LIN {X 0,Y 616.016,Z 683.652,A -85,B 0,C 180,E1 29122.379,E2 29122.379} C_VEL
LIN {X 0,Y 617.28,Z 685.528,A -85,B 0,C 180,E1 29121.476,E2 29121.476} C_VEL
LIN {X 0,Y 619.5,Z 690.288,A -85,B 0,C 180,E1 29120.03,E2 29120.03} C_VEL
LIN {X 0,Y 621.765,Z 695.272,A -85,B 0,C 180,E1 29118.873,E2 29118.873} C_VEL
LIN {X 0,Y 624.795,Z 702.465,A -85,B 0,C 180,E1 29117.519,E2 29117.519} C_VEL
LIN {X 0,Y 628.158,Z 711.521,A -85,B 0,C 180,E1 29116.158,E2 29116.158} C_VEL
LIN {X 0,Y 622.39,Z 748.268,A -85,B 0,C 180,E1 29113.628,E2 29113.628} C_VEL
LIN {X 0,Y 618.399,Z 786.592,A -85,B 0,C 180,E1 29111.107,E2 29111.107} C_VEL
LIN {X 0,Y 618.395,Z 807.892,A -85,B 0,C 180,E1 29109.637,E2 29109.637} C_VEL
LIN {X 0,Y 620.24,Z 824.543,A -85,B 0,C 180,E1 29108.419,E2 29108.419} C_VEL
LIN {X 0,Y 623.991,Z 840.098,A -85,B 0,C 180,E1 29107.212,E2 29107.212} C_VEL
LIN {X 0,Y 629.828,Z 854.618,A -85,B 0,C 180,E1 29106.015,E2 29106.015} C_VEL
LIN {X 0,Y 636.961,Z 866.767,A -85,B 0,C 180,E1 29104.955,E2 29104.955} C_VEL
LIN {X 0,Y 645.236,Z 877.236,A -85,B 0,C 180,E1 29103.997,E2 29103.997} C_VEL
LIN {X 0,Y 655.85,Z 887.383,A -85,B 0,C 180,E1 29103.016,E2 29103.016} C_VEL
LIN {X 0,Y 667.322,Z 895.733,A -85,B 0,C 180,E1 29102.159,E2 29102.159} C_VEL
LIN {X 0,Y 672.025,Z 898.736,A -85,B 0,C 180,E1 29101.844,E2 29101.844} C_VEL
LIN {X 0,Y 649.338,Z 931.659,A -85,B 0,C 180,E1 29100.95,E2 29100.95} C_VEL
LIN {X 0,Y 638.123,Z 950.658,A -85,B 0,C 180,E1 29100.351,E2 29100.351} C_VEL
LIN {X 0,Y 630.355,Z 966.843,A -85,B 0,C 180,E1 29099.766,E2 29099.766} C_VEL
LIN {X 0,Y 626.313,Z 976.356,A -85,B 0,C 180,E1 29099.399,E2 29099.399} C_VEL
LIN {X 0,Y 619.977,Z 991.013,A -85,B 0,C 180,E1 29098.829,E2 29098.829} C_VEL
LIN {X 0,Y 614.207,Z 1008.828,A -85,B 0,C 180,E1 29098.082,E2 29098.082} C_VEL
LIN {X 0,Y 612.745,Z 1027.64,A -85,B 0,C 180,E1 29097.893,E2 29097.893} C_VEL
LIN {X 0,Y 612.102,Z 1064.345,A -85,B 0,C 180,E1 29097.385,E2 29097.385} C_VEL
LIN {X 0,Y 611.36,Z 1085.866,A -85,B 0,C 180,E1 29096.927,E2 29096.927} C_VEL
LIN {X 0,Y 610.423,Z 1107.35,A -85,B 0,C 180,E1 29096.299,E2 29096.299} C_VEL
LIN {X 0,Y 609.333,Z 1128.576,A -85,B 0,C 180,E1 29095.507,E2 29095.507} C_VEL
LIN {X 0,Y 608.179,Z 1148.795,A -85,B 0,C 180,E1 29094.577,E2 29094.577} C_VEL
LIN {X 0,Y 606.971,Z 1168.175,A -85,B 0,C 180,E1 29093.492,E2 29093.492} C_VEL
LIN {X 0,Y 605.739,Z 1186.859,A -85,B 0,C 180,E1 29092.26,E2 29092.26} C_VEL
LIN {X 0,Y 604.616,Z 1204.162,A -85,B 0,C 180,E1 29090.927,E2 29090.927} C_VEL
LIN {X 0,Y 603.528,Z 1220.54,A -85,B 0,C 180,E1 29089.45,E2 29089.45} C_VEL
LIN {X 0,Y 602.577,Z 1235.528,A -85,B 0,C 180,E1 29087.876,E2 29087.876} C_VEL
LIN {X 0,Y 601.792,Z 1249.417,A -85,B 0,C 180,E1 29086.186,E2 29086.186} C_VEL
LIN {X 0,Y 601.099,Z 1262.801,A -85,B 0,C 180,E1 29084.251,E2 29084.251} C_VEL
LIN {X 0,Y 600.679,Z 1273.278,A -85,B 0,C 180,E1 29082.496,E2 29082.496} C_VEL
LIN {X 0,Y 600.389,Z 1281.271,A -85,B 0,C 180,E1 29080.943,E2 29080.943} C_VEL
LIN {X 0,Y 600.168,Z 1289.619,A -85,B 0,C 180,E1 29079.008,E2 29079.008} C_VEL
LIN {X 0,Y 600.052,Z 1295.993,A -85,B 0,C 180,E1 29077.082,E2 29077.082} C_VEL
LIN {X 0,Y 599.998,Z 1300.183,A -85,B 0,C 180,E1 29075.449,E2 29075.449} C_VEL
LIN {X 0,Y 599.968,Z 1303.25,A -85,B 0,C 180,E1 29073.821,E2 29073.821} C_VEL
LIN {X 0,Y 599.962,Z 1305.145,A -85,B 0,C 180,E1 29072.291,E2 29072.291} C_VEL
LIN {X 0,Y 599.962,Z 1306.122,A -85,B 0,C 180,E1 29070.667,E2 29070.667} C_VEL
LIN {X 0,Y 599.969,Z 1306.047,A -85,B 0,C 180,E1 29069.044,E2 29069.044} C_VEL
LIN {X 0,Y 599.968,Z 1304.572,A -85,B 0,C 180,E1 29067.037,E2 29067.037} C_VEL
LIN {X 0,Y 599.975,Z 1301.11,A -85,B 0,C 180,E1 29064.931,E2 29064.931} C_VEL
LIN {X 0,Y 600.018,Z 1296.951,A -85,B 0,C 180,E1 29063.204,E2 29063.204} C_VEL
LIN {X 0,Y 600.122,Z 1291.846,A -85,B 0,C 180,E1 29061.568,E2 29061.568} C_VEL
LIN {X 0,Y 600.293,Z 1284.34,A -85,B 0,C 180,E1 29059.635,E2 29059.635} C_VEL
LIN {X 0,Y 600.621,Z 1274.844,A -85,B 0,C 180,E1 29057.695,E2 29057.695} C_VEL
LIN {X 0,Y 600.987,Z 1265.818,A -85,B 0,C 180,E1 29056.137,E2 29056.137} C_VEL
LIN {X 0,Y 601.5,Z 1255.377,A -85,B 0,C 180,E1 29054.574,E2 29054.574} C_VEL
LIN {X 0,Y 602.228,Z 1241.71,A -85,B 0,C 180,E1 29052.809,E2 29052.809} C_VEL
LIN {X 0,Y 603.089,Z 1227.052,A -85,B 0,C 180,E1 29051.208,E2 29051.208} C_VEL
LIN {X 0,Y 603.966,Z 1212.919,A -85,B 0,C 180,E1 29049.857,E2 29049.857} C_VEL
LIN {X 0,Y 605.154,Z 1194.406,A -85,B 0,C 180,E1 29048.327,E2 29048.327} C_VEL
LIN {X 0,Y 606.276,Z 1176.824,A -85,B 0,C 180,E1 29047.093,E2 29047.093} C_VEL
LIN {X 0,Y 607.501,Z 1156.987,A -85,B 0,C 180,E1 29045.908,E2 29045.908} C_VEL
LIN {X 0,Y 608.668,Z 1137.497,A -85,B 0,C 180,E1 29044.922,E2 29044.922} C_VEL
LIN {X 0,Y 609.771,Z 1116.588,A -85,B 0,C 180,E1 29044.063,E2 29044.063} C_VEL
LIN {X 0,Y 610.873,Z 1093.442,A -85,B 0,C 180,E1 29043.306,E2 29043.306} C_VEL
LIN {X 0,Y 611.749,Z 1071.492,A -85,B 0,C 180,E1 29042.763,E2 29042.763} C_VEL
LIN {X 0,Y 612.378,Z 1049.209,A -85,B 0,C 180,E1 29042.388,E2 29042.388} C_VEL
LIN {X 0,Y 613.089,Z 1019.395,A -85,B 0,C 180,E1 29042.016,E2 29042.016} C_VEL
LIN {X 0,Y 613.475,Z 1017.129,A -85,B 0,C 180,E1 29041.951,E2 29041.951} C_VEL
LIN {X 0,Y 619.742,Z 996.837,A -85,B 0,C 180,E1 29041.051,E2 29041.051} C_VEL
LIN {X 0,Y 625.666,Z 982.108,A -85,B 0,C 180,E1 29040.46,E2 29040.46} C_VEL
LIN {X 0,Y 629.987,Z 972.662,A -85,B 0,C 180,E1 29040.107,E2 29040.107} C_VEL
LIN {X 0,Y 636.958,Z 957.167,A -85,B 0,C 180,E1 29039.532,E2 29039.532} C_VEL
LIN {X 0,Y 647.358,Z 938.566,A -85,B 0,C 180,E1 29038.942,E2 29038.942} C_VEL
LIN {X 0,Y 663.158,Z 914.467,A -85,B 0,C 180,E1 29038.305,E2 29038.305} C_VEL
LIN {X 0,Y 672.936,Z 899.902,A -85,B 0,C 180,E1 29037.949,E2 29037.949} C_VEL
LIN {X 0,Y 660.637,Z 891.93,A -85,B 0,C 180,E1 29036.982,E2 29036.982} C_VEL
LIN {X 0,Y 650.17,Z 882.751,A -85,B 0,C 180,E1 29035.989,E2 29035.989} C_VEL
LIN {X 0,Y 641.576,Z 872.759,A -85,B 0,C 180,E1 29035.003,E2 29035.003} C_VEL
LIN {X 0,Y 634,Z 860.886,A -85,B 0,C 180,E1 29033.928,E2 29033.928} C_VEL
LIN {X 0,Y 627.838,Z 847.084,A -85,B 0,C 180,E1 29032.778,E2 29032.778} C_VEL
LIN {X 0,Y 623.551,Z 832.289,A -85,B 0,C 180,E1 29031.641,E2 29031.641} C_VEL
LIN {X 0,Y 620.905,Z 815.947,A -85,B 0,C 180,E1 29030.477,E2 29030.477} C_VEL
LIN {X 0,Y 619.883,Z 794.864,A -85,B 0,C 180,E1 29029.088,E2 29029.088} C_VEL
LIN {X 0,Y 621.669,Z 759.114,A -85,B 0,C 180,E1 29026.904,E2 29026.904} C_VEL
LIN {X 0,Y 625.012,Z 710.924,A -85,B 0,C 180,E1 29023.944,E2 29023.944} C_VEL
LIN {X 0,Y 613.302,Z 684.566,A -85,B 0,C 180,E1 29021.198,E2 29021.198} C_VEL
LIN {X 0,Y 604.079,Z 664.832,A -85,B 0,C 180,E1 29018.976,E2 29018.976} C_VEL
LIN {X 0,Y 602.19,Z 660.891,A -85,B 0,C 180,E1 29018.511,E2 29018.511} C_VEL
LIN {X 0,Y 601.247,Z 658.443,A -85,B 0,C 180,E1 29018.233,E2 29018.233} C_VEL
LIN {X 0,Y 602.826,Z 661.813,A -85,B 0,C 180,E1 29017.703,E2 29017.703} C_VEL
LIN {X 0,Y 606.74,Z 670.074,A -85,B 0,C 180,E1 29016.465,E2 29016.465} C_VEL
LIN {X 0,Y 611.287,Z 682.203,A -85,B 0,C 180,E1 29014.883,E2 29014.883} C_VEL
LIN {X 0,Y 615.347,Z 696.845,A -85,B 0,C 180,E1 29013.192,E2 29013.192} C_VEL
LIN {X 0,Y 615.108,Z 709.007,A -85,B 0,C 180,E1 29012.165,E2 29012.165} C_VEL
LIN {X 0,Y 619.393,Z 729.053,A -85,B 0,C 180,E1 29011.452,E2 29011.452} C_VEL
LIN {X 0,Y 615.849,Z 837.863,A -85,B 0,C 180,E1 29009.755,E2 29009.755} C_VEL
LIN {X 0,Y 613.356,Z 948.464,A -85,B 0,C 180,E1 29008.178,E2 29008.178} C_VEL
LIN {X 0,Y 612.308,Z 1010.047,A -85,B 0,C 180,E1 29007.333,E2 29007.333} C_VEL
LIN {X 0,Y 611.653,Z 1032.255,A -85,B 0,C 180,E1 29006.862,E2 29006.862} C_VEL
LIN {X 0,Y 610.807,Z 1054.79,A -85,B 0,C 180,E1 29006.205,E2 29006.205} C_VEL
LIN {X 0,Y 609.858,Z 1075.299,A -85,B 0,C 180,E1 29005.44,E2 29005.44} C_VEL
LIN {X 0,Y 608.759,Z 1095.579,A -85,B 0,C 180,E1 29004.501,E2 29004.501} C_VEL
LIN {X 0,Y 607.572,Z 1114.908,A -85,B 0,C 180,E1 29003.418,E2 29003.418} C_VEL
LIN {X 0,Y 606.32,Z 1134.142,A -85,B 0,C 180,E1 29002.137,E2 29002.137} C_VEL
LIN {X 0,Y 605.157,Z 1151.119,A -85,B 0,C 180,E1 29000.808,E2 29000.808} C_VEL
LIN {X 0,Y 604.031,Z 1167.132,A -85,B 0,C 180,E1 28999.334,E2 28999.334} C_VEL
LIN {X 0,Y 603.018,Z 1181.706,A -85,B 0,C 180,E1 28997.764,E2 28997.764} C_VEL
LIN {X 0,Y 602.139,Z 1194.991,A -85,B 0,C 180,E1 28996.1,E2 28996.1} C_VEL
LIN {X 0,Y 601.407,Z 1206.895,A -85,B 0,C 180,E1 28994.343,E2 28994.343} C_VEL
LIN {X 0,Y 600.831,Z 1217.366,A -85,B 0,C 180,E1 28992.494,E2 28992.494} C_VEL
LIN {X 0,Y 600.415,Z 1226.896,A -85,B 0,C 180,E1 28990.458,E2 28990.458} C_VEL
LIN {X 0,Y 600.155,Z 1234.212,A -85,B 0,C 180,E1 28988.527,E2 28988.527} C_VEL
LIN {X 0,Y 600.015,Z 1240.016,A -85,B 0,C 180,E1 28986.507,E2 28986.507} C_VEL
LIN {X 0,Y 599.947,Z 1244.377,A -85,B 0,C 180,E1 28984.397,E2 28984.397} C_VEL
LIN {X 0,Y 599.919,Z 1247.007,A -85,B 0,C 180,E1 28982.388,E2 28982.388} C_VEL
LIN {X 0,Y 599.919,Z 1248.01,A -85,B 0,C 180,E1 28980.382,E2 28980.382} C_VEL
LIN {X 0,Y 599.926,Z 1247.442,A -85,B 0,C 180,E1 28978.185,E2 28978.185} C_VEL
LIN {X 0,Y 599.93,Z 1245.409,A -85,B 0,C 180,E1 28976.177,E2 28976.177} C_VEL
LIN {X 0,Y 599.976,Z 1241.714,A -85,B 0,C 180,E1 28974.165,E2 28974.165} C_VEL
LIN {X 0,Y 600.089,Z 1236.152,A -85,B 0,C 180,E1 28972.051,E2 28972.051} C_VEL
LIN {X 0,Y 600.308,Z 1229.115,A -85,B 0,C 180,E1 28970.025,E2 28970.025} C_VEL
LIN {X 0,Y 600.668,Z 1220.605,A -85,B 0,C 180,E1 28968.088,E2 28968.088} C_VEL
LIN {X 0,Y 601.196,Z 1210.173,A -85,B 0,C 180,E1 28966.143,E2 28966.143} C_VEL
LIN {X 0,Y 601.948,Z 1197.606,A -85,B 0,C 180,E1 28964.192,E2 28964.192} C_VEL
LIN {X 0,Y 602.807,Z 1184.861,A -85,B 0,C 180,E1 28962.511,E2 28962.511} C_VEL
LIN {X 0,Y 603.847,Z 1170.11,A -85,B 0,C 180,E1 28960.861,E2 28960.861} C_VEL
LIN {X 0,Y 605.021,Z 1154.227,A -85,B 0,C 180,E1 28959.339,E2 28959.339} C_VEL
LIN {X 0,Y 606.296,Z 1136.887,A -85,B 0,C 180,E1 28957.913,E2 28957.913} C_VEL
LIN {X 0,Y 607.621,Z 1118.65,A -85,B 0,C 180,E1 28956.635,E2 28956.635} C_VEL
LIN {X 0,Y 608.908,Z 1099.293,A -85,B 0,C 180,E1 28955.499,E2 28955.499} C_VEL
LIN {X 0,Y 610.13,Z 1079.481,A -85,B 0,C 180,E1 28954.526,E2 28954.526} C_VEL
LIN {X 0,Y 611.266,Z 1058.642,A -85,B 0,C 180,E1 28953.686,E2 28953.686} C_VEL
LIN {X 0,Y 612.254,Z 1037.215,A -85,B 0,C 180,E1 28953.008,E2 28953.008} C_VEL
LIN {X 0,Y 612.996,Z 1015.392,A -85,B 0,C 180,E1 28952.494,E2 28952.494} C_VEL
LIN {X 0,Y 613.627,Z 988.931,A -85,B 0,C 180,E1 28952.078,E2 28952.078} C_VEL
LIN {X 0,Y 617.321,Z 776.467,A -85,B 0,C 180,E1 28949.286,E2 28949.286} C_VEL
LIN {X 0,Y 618.112,Z 728.534,A -85,B 0,C 180,E1 28948.627,E2 28948.627} C_VEL
LIN {X 0,Y 613.662,Z 708.816,A -85,B 0,C 180,E1 28948.086,E2 28948.086} C_VEL
LIN {X 0,Y 612.342,Z 704.037,A -85,B 0,C 180,E1 28947.867,E2 28947.867} C_VEL
LIN {X 0,Y 610.115,Z 698.563,A -85,B 0,C 180,E1 28947.392,E2 28947.392} C_VEL
LIN {X 0,Y 604.965,Z 691.045,A -85,B 0,C 180,E1 28946.41,E2 28946.41} C_VEL
LIN {X 0,Y 602.343,Z 686.435,A -85,B 0,C 180,E1 28945.826,E2 28945.826} C_VEL
LIN {X 0,Y 602.1,Z 685.7,A -85,B 0,C 180,E1 28945.744,E2 28945.744} C_VEL
LIN {X 0,Y 594.907,Z 664.107,A -85,B 0,C 180,E1 28943.295,E2 28943.295} C_VEL
LIN {X 0,Y 593.182,Z 658.781,A -85,B 0,C 180,E1 28942.671,E2 28942.671} C_VEL
LIN {X 0,Y 593.182,Z 658.78,A -85,B 0,C 180,E1 28939.485,E2 28939.485} C_VEL
LIN {X 0,Y 593.183,Z 658.781,A -85,B 0,C 180,E1 28936.282,E2 28936.282} C_VEL
LIN {X 0,Y 593.191,Z 658.778,A -85,B 0,C 180,E1 28933.054,E2 28933.054} C_VEL
LIN {X 0,Y 593.185,Z 658.778,A -85,B 0,C 180,E1 28929.833,E2 28929.833} C_VEL
LIN {X 0,Y 593.187,Z 658.774,A -85,B 0,C 180,E1 28926.636,E2 28926.636} C_VEL
LIN {X 0,Y 593.199,Z 658.772,A -85,B 0,C 180,E1 28923.274,E2 28923.274} C_VEL
LIN {X 0,Y 593.188,Z 658.773,A -85,B 0,C 180,E1 28919.931,E2 28919.931} C_VEL
LIN {X 0,Y 593.184,Z 658.777,A -85,B 0,C 180,E1 28916.698,E2 28916.698} C_VEL
LIN {X 0,Y 593.198,Z 658.78,A -85,B 0,C 180,E1 28913.442,E2 28913.442} C_VEL
LIN {X 0,Y 593.2,Z 658.781,A -85,B 0,C 180,E1 28910.113,E2 28910.113} C_VEL
LIN {X 0,Y 593.189,Z 658.777,A -85,B 0,C 180,E1 28906.855,E2 28906.855} C_VEL
LIN {X 0,Y 593.195,Z 658.771,A -85,B 0,C 180,E1 28903.551,E2 28903.551} C_VEL
LIN {X 0,Y 593.189,Z 658.774,A -85,B 0,C 180,E1 28900.196,E2 28900.196} C_VEL
LIN {X 0,Y 593.184,Z 658.776,A -85,B 0,C 180,E1 28896.972,E2 28896.972} C_VEL
LIN {X 0,Y 593.181,Z 658.776,A -85,B 0,C 180,E1 28893.71,E2 28893.71} C_VEL
LIN {X 0,Y 593.197,Z 658.775,A -85,B 0,C 180,E1 28890.484,E2 28890.484} C_VEL
LIN {X 0,Y 593.183,Z 658.779,A -85,B 0,C 180,E1 28887.296,E2 28887.296} C_VEL
LIN {X 0,Y 593.183,Z 658.776,A -85,B 0,C 180,E1 28884.1,E2 28884.1} C_VEL
LIN {X 0,Y 593.185,Z 658.776,A -85,B 0,C 180,E1 28880.885,E2 28880.885} C_VEL
LIN {X 0,Y 593.199,Z 658.776,A -85,B 0,C 180,E1 28877.542,E2 28877.542} C_VEL
LIN {X 0,Y 593.194,Z 658.78,A -85,B 0,C 180,E1 28874.255,E2 28874.255} C_VEL
LIN {X 0,Y 593.202,Z 658.781,A -85,B 0,C 180,E1 28871.017,E2 28871.017} C_VEL
LIN {X 0,Y 593.181,Z 658.78,A -85,B 0,C 180,E1 28867.732,E2 28867.732} C_VEL
LIN {X 0,Y 593.182,Z 658.774,A -85,B 0,C 180,E1 28864.545,E2 28864.545} C_VEL
LIN {X 0,Y 593.181,Z 658.778,A -85,B 0,C 180,E1 28861.4,E2 28861.4} C_VEL
LIN {X 0,Y 593.188,Z 658.77,A -85,B 0,C 180,E1 28858.272,E2 28858.272} C_VEL
LIN {X 0,Y 593.187,Z 658.777,A -85,B 0,C 180,E1 28855.007,E2 28855.007} C_VEL
LIN {X 0,Y 593.187,Z 658.779,A -85,B 0,C 180,E1 28851.767,E2 28851.767} C_VEL
LIN {X 0,Y 593.197,Z 658.77,A -85,B 0,C 180,E1 28848.453,E2 28848.453} C_VEL
LIN {X 0,Y 593.208,Z 658.843,A -85,B 0,C 180,E1 28846.312,E2 28846.312} C_VEL
LIN {X 0,Y 602.946,Z 685.523,A -85,B 0,C 180,E1 28843.358,E2 28843.358} C_VEL
LIN {X 0,Y 608.157,Z 701.222,A -85,B 0,C 180,E1 28841.72,E2 28841.72} C_VEL
LIN {X 0,Y 606.076,Z 738.611,A -85,B 0,C 180,E1 28838.823,E2 28838.823} C_VEL
LIN {X 0,Y 603.739,Z 781.028,A -85,B 0,C 180,E1 28835.596,E2 28835.596} C_VEL
LIN {X 0,Y 601.529,Z 824.766,A -85,B 0,C 180,E1 28832.304,E2 28832.304} C_VEL
LIN {X 0,Y 599.443,Z 871.743,A -85,B 0,C 180,E1 28828.82,E2 28828.82} C_VEL
LIN {X 0,Y 598.38,Z 900.943,A -85,B 0,C 180,E1 28826.705,E2 28826.705} C_VEL
LIN {X 0,Y 599.197,Z 909.396,A -85,B 0,C 180,E1 28826.545,E2 28826.545} C_VEL
LIN {X 0,Y 596.797,Z 1045.223,A -85,B 0,C 180,E1 28824.486,E2 28824.486} C_VEL
LIN {X 0,Y 596.512,Z 1062.31,A -85,B 0,C 180,E1 28824.037,E2 28824.037} C_VEL
LIN {X 0,Y 596.1,Z 1078.016,A -85,B 0,C 180,E1 28823.438,E2 28823.438} C_VEL
LIN {X 0,Y 595.577,Z 1093.217,A -85,B 0,C 180,E1 28822.662,E2 28822.662} C_VEL
LIN {X 0,Y 595.037,Z 1107.189,A -85,B 0,C 180,E1 28821.748,E2 28821.748} C_VEL
LIN {X 0,Y 594.463,Z 1120.603,A -85,B 0,C 180,E1 28820.643,E2 28820.643} C_VEL
LIN {X 0,Y 593.958,Z 1132.014,A -85,B 0,C 180,E1 28819.471,E2 28819.471} C_VEL
LIN {X 0,Y 593.494,Z 1142.261,A -85,B 0,C 180,E1 28818.161,E2 28818.161} C_VEL
LIN {X 0,Y 593.13,Z 1150.907,A -85,B 0,C 180,E1 28816.767,E2 28816.767} C_VEL
LIN {X 0,Y 592.858,Z 1158.098,A -85,B 0,C 180,E1 28815.254,E2 28815.254} C_VEL
LIN {X 0,Y 592.705,Z 1163.31,A -85,B 0,C 180,E1 28813.761,E2 28813.761} C_VEL
LIN {X 0,Y 592.618,Z 1167.102,A -85,B 0,C 180,E1 28812.077,E2 28812.077} C_VEL
LIN {X 0,Y 592.598,Z 1168.846,A -85,B 0,C 180,E1 28810.5,E2 28810.5} C_VEL
LIN {X 0,Y 592.649,Z 1168.776,A -85,B 0,C 180,E1 28808.832,E2 28808.832} C_VEL
LIN {X 0,Y 592.748,Z 1166.971,A -85,B 0,C 180,E1 28807.268,E2 28807.268} C_VEL
LIN {X 0,Y 592.934,Z 1163.121,A -85,B 0,C 180,E1 28805.613,E2 28805.613} C_VEL
LIN {X 0,Y 593.212,Z 1158.017,A -85,B 0,C 180,E1 28804.156,E2 28804.156} C_VEL
LIN {X 0,Y 593.624,Z 1150.545,A -85,B 0,C 180,E1 28802.607,E2 28802.607} C_VEL
LIN {X 0,Y 594.127,Z 1142.09,A -85,B 0,C 180,E1 28801.254,E2 28801.254} C_VEL
LIN {X 0,Y 594.765,Z 1131.36,A -85,B 0,C 180,E1 28799.904,E2 28799.904} C_VEL
LIN {X 0,Y 595.414,Z 1119.883,A -85,B 0,C 180,E1 28798.749,E2 28798.749} C_VEL
LIN {X 0,Y 596.122,Z 1106.14,A -85,B 0,C 180,E1 28797.645,E2 28797.645} C_VEL
LIN {X 0,Y 596.732,Z 1092.506,A -85,B 0,C 180,E1 28796.782,E2 28796.782} C_VEL
LIN {X 0,Y 597.333,Z 1076.957,A -85,B 0,C 180,E1 28796.017,E2 28796.017} C_VEL
LIN {X 0,Y 597.748,Z 1061.003,A -85,B 0,C 180,E1 28795.443,E2 28795.443} C_VEL
LIN {X 0,Y 598.009,Z 1044.535,A -85,B 0,C 180,E1 28795.039,E2 28795.039} C_VEL
LIN {X 0,Y 602.648,Z 910.21,A -85,B 0,C 180,E1 28792.564,E2 28792.564} C_VEL
LIN {X 0,Y 606.159,Z 864.366,A -85,B 0,C 180,E1 28788.925,E2 28788.925} C_VEL
LIN {X 0,Y 610.133,Z 822.222,A -85,B 0,C 180,E1 28785.479,E2 28785.479} C_VEL
LIN {X 0,Y 614.922,Z 781.575,A -85,B 0,C 180,E1 28782.053,E2 28782.053} C_VEL
LIN {X 0,Y 620.198,Z 745.319,A -85,B 0,C 180,E1 28778.879,E2 28778.879} C_VEL
LIN {X 0,Y 623.445,Z 723.04,A -85,B 0,C 180,E1 28776.773,E2 28776.773} C_VEL
LIN {X 0,Y 619.661,Z 711.696,A -85,B 0,C 180,E1 28774.786,E2 28774.786} C_VEL
LIN {X 0,Y 616.192,Z 702.269,A -85,B 0,C 180,E1 28772.768,E2 28772.768} C_VEL
LIN {X 0,Y 614.012,Z 697.274,A -85,B 0,C 180,E1 28771.395,E2 28771.395} C_VEL
LIN {X 0,Y 612.775,Z 694.186,A -85,B 0,C 180,E1 28770.422,E2 28770.422} C_VEL
LIN {X 0,Y 611.373,Z 690.559,A -85,B 0,C 180,E1 28768.976,E2 28768.976} C_VEL
LIN {X 0,Y 610.067,Z 687.576,A -85,B 0,C 180,E1 28766.922,E2 28766.922} C_VEL
LIN {X 0,Y 610.098,Z 686.717,A -85,B 0,C 180,E1 28765.796,E2 28765.796} C_VEL
LIN {X 0,Y 610.364,Z 687.182,A -85,B 0,C 180,E1 28764.324,E2 28764.324} C_VEL
LIN {X 0,Y 611.582,Z 690.406,A -85,B 0,C 180,E1 28762.304,E2 28762.304} C_VEL
LIN {X 0,Y 612.597,Z 692.036,A -85,B 0,C 180,E1 28761.547,E2 28761.547} C_VEL
LIN {X 0,Y 614.682,Z 696.587,A -85,B 0,C 180,E1 28760.14,E2 28760.14} C_VEL
LIN {X 0,Y 616.962,Z 701.817,A -85,B 0,C 180,E1 28758.901,E2 28758.901} C_VEL
LIN {X 0,Y 620.027,Z 709.43,A -85,B 0,C 180,E1 28757.472,E2 28757.472} C_VEL
LIN {X 0,Y 622.203,Z 715.955,A -85,B 0,C 180,E1 28756.492,E2 28756.492} C_VEL
LIN {X 0,Y 616.047,Z 752.427,A -85,B 0,C 180,E1 28753.934,E2 28753.934} C_VEL
LIN {X 0,Y 611.893,Z 788.668,A -85,B 0,C 180,E1 28751.498,E2 28751.498} C_VEL
LIN {X 0,Y 611.616,Z 809.418,A -85,B 0,C 180,E1 28750.036,E2 28750.036} C_VEL
LIN {X 0,Y 613.216,Z 826.516,A -85,B 0,C 180,E1 28748.763,E2 28748.763} C_VEL
LIN {X 0,Y 616.826,Z 842.664,A -85,B 0,C 180,E1 28747.487,E2 28747.487} C_VEL
LIN {X 0,Y 622.441,Z 857.371,A -85,B 0,C 180,E1 28746.253,E2 28746.253} C_VEL
LIN {X 0,Y 629.001,Z 869.22,A -85,B 0,C 180,E1 28745.206,E2 28745.206} C_VEL
LIN {X 0,Y 637.764,Z 880.886,A -85,B 0,C 180,E1 28744.126,E2 28744.126} C_VEL
LIN {X 0,Y 648.799,Z 891.796,A -85,B 0,C 180,E1 28743.061,E2 28743.061} C_VEL
LIN {X 0,Y 660.295,Z 900.467,A -85,B 0,C 180,E1 28742.167,E2 28742.167} C_VEL
LIN {X 0,Y 661.725,Z 901.682,A -85,B 0,C 180,E1 28742.054,E2 28742.054} C_VEL
LIN {X 0,Y 642.342,Z 930.073,A -85,B 0,C 180,E1 28741.285,E2 28741.285} C_VEL
LIN {X 0,Y 631.045,Z 949.308,A -85,B 0,C 180,E1 28740.676,E2 28740.676} C_VEL
LIN {X 0,Y 623.284,Z 965.503,A -85,B 0,C 180,E1 28740.085,E2 28740.085} C_VEL
LIN {X 0,Y 619.197,Z 975.007,A -85,B 0,C 180,E1 28739.717,E2 28739.717} C_VEL
LIN {X 0,Y 612.523,Z 990.547,A -85,B 0,C 180,E1 28739.106,E2 28739.106} C_VEL
LIN {X 0,Y 607.229,Z 1006.828,A -85,B 0,C 180,E1 28738.423,E2 28738.423} C_VEL
LIN {X 0,Y 605.497,Z 1027.168,A -85,B 0,C 180,E1 28738.218,E2 28738.218} C_VEL
LIN {X 0,Y 604.811,Z 1063.902,A -85,B 0,C 180,E1 28737.703,E2 28737.703} C_VEL
LIN {X 0,Y 604.03,Z 1085.343,A -85,B 0,C 180,E1 28737.241,E2 28737.241} C_VEL
LIN {X 0,Y 603.05,Z 1106.508,A -85,B 0,C 180,E1 28736.619,E2 28736.619} C_VEL
LIN {X 0,Y 601.949,Z 1127.147,A -85,B 0,C 180,E1 28735.849,E2 28735.849} C_VEL
LIN {X 0,Y 600.678,Z 1148.18,A -85,B 0,C 180,E1 28734.877,E2 28734.877} C_VEL
LIN {X 0,Y 599.375,Z 1168.01,A -85,B 0,C 180,E1 28733.756,E2 28733.756} C_VEL
LIN {X 0,Y 598.062,Z 1186.665,A -85,B 0,C 180,E1 28732.509,E2 28732.509} C_VEL
LIN {X 0,Y 596.881,Z 1203.95,A -85,B 0,C 180,E1 28731.16,E2 28731.16} C_VEL
LIN {X 0,Y 595.735,Z 1220.166,A -85,B 0,C 180,E1 28729.679,E2 28729.679} C_VEL
LIN {X 0,Y 594.741,Z 1234.867,A -85,B 0,C 180,E1 28728.119,E2 28728.119} C_VEL
LIN {X 0,Y 593.921,Z 1248.657,A -85,B 0,C 180,E1 28726.428,E2 28726.428} C_VEL
LIN {X 0,Y 593.199,Z 1261.697,A -85,B 0,C 180,E1 28724.544,E2 28724.544} C_VEL
LIN {X 0,Y 592.718,Z 1272.532,A -85,B 0,C 180,E1 28722.667,E2 28722.667} C_VEL
LIN {X 0,Y 592.358,Z 1282.099,A -85,B 0,C 180,E1 28720.699,E2 28720.699} C_VEL
LIN {X 0,Y 592.172,Z 1290.272,A -85,B 0,C 180,E1 28718.642,E2 28718.642} C_VEL
LIN {X 0,Y 592.074,Z 1295.548,A -85,B 0,C 180,E1 28716.983,E2 28716.983} C_VEL
LIN {X 0,Y 592.034,Z 1299.653,A -85,B 0,C 180,E1 28715.328,E2 28715.328} C_VEL
LIN {X 0,Y 592.012,Z 1302.63,A -85,B 0,C 180,E1 28713.678,E2 28713.678} C_VEL
LIN {X 0,Y 592.013,Z 1304.695,A -85,B 0,C 180,E1 28711.838,E2 28711.838} C_VEL
LIN {X 0,Y 592.003,Z 1305.34,A -85,B 0,C 180,E1 28709.612,E2 28709.612} C_VEL
LIN {X 0,Y 592.004,Z 1304.482,A -85,B 0,C 180,E1 28707.869,E2 28707.869} C_VEL
LIN {X 0,Y 592.001,Z 1302.586,A -85,B 0,C 180,E1 28706.222,E2 28706.222} C_VEL
LIN {X 0,Y 592.02,Z 1299.607,A -85,B 0,C 180,E1 28704.572,E2 28704.572} C_VEL
LIN {X 0,Y 592.075,Z 1295.244,A -85,B 0,C 180,E1 28702.82,E2 28702.82} C_VEL
LIN {X 0,Y 592.197,Z 1288.131,A -85,B 0,C 180,E1 28700.671,E2 28700.671} C_VEL
LIN {X 0,Y 592.419,Z 1280.193,A -85,B 0,C 180,E1 28698.807,E2 28698.807} C_VEL
LIN {X 0,Y 592.746,Z 1271.697,A -85,B 0,C 180,E1 28697.133,E2 28697.133} C_VEL
LIN {X 0,Y 593.283,Z 1259.784,A -85,B 0,C 180,E1 28695.156,E2 28695.156} C_VEL
LIN {X 0,Y 593.93,Z 1247.612,A -85,B 0,C 180,E1 28693.469,E2 28693.469} C_VEL
LIN {X 0,Y 594.649,Z 1235.271,A -85,B 0,C 180,E1 28691.976,E2 28691.976} C_VEL
LIN {X 0,Y 595.642,Z 1219.824,A -85,B 0,C 180,E1 28690.346,E2 28690.346} C_VEL
LIN {X 0,Y 596.727,Z 1203.454,A -85,B 0,C 180,E1 28688.883,E2 28688.883} C_VEL
LIN {X 0,Y 597.794,Z 1187.553,A -85,B 0,C 180,E1 28687.638,E2 28687.638} C_VEL
LIN {X 0,Y 599.102,Z 1168.023,A -85,B 0,C 180,E1 28686.334,E2 28686.334} C_VEL
LIN {X 0,Y 600.335,Z 1148.673,A -85,B 0,C 180,E1 28685.235,E2 28685.235} C_VEL
LIN {X 0,Y 601.565,Z 1128.125,A -85,B 0,C 180,E1 28684.275,E2 28684.275} C_VEL
LIN {X 0,Y 602.746,Z 1106.285,A -85,B 0,C 180,E1 28683.443,E2 28683.443} C_VEL
LIN {X 0,Y 603.799,Z 1084.344,A -85,B 0,C 180,E1 28682.786,E2 28682.786} C_VEL
LIN {X 0,Y 604.619,Z 1062.444,A -85,B 0,C 180,E1 28682.312,E2 28682.312} C_VEL
LIN {X 0,Y 605.299,Z 1029.223,A -85,B 0,C 180,E1 28681.833,E2 28681.833} C_VEL
LIN {X 0,Y 605.997,Z 1017.171,A -85,B 0,C 180,E1 28681.681,E2 28681.681} C_VEL
LIN {X 0,Y 611.962,Z 997.847,A -85,B 0,C 180,E1 28680.808,E2 28680.808} C_VEL
LIN {X 0,Y 618.069,Z 982.25,A -85,B 0,C 180,E1 28680.167,E2 28680.167} C_VEL
LIN {X 0,Y 623.529,Z 970.242,A -85,B 0,C 180,E1 28679.712,E2 28679.712} C_VEL
LIN {X 0,Y 631.066,Z 953.948,A -85,B 0,C 180,E1 28679.111,E2 28679.111} C_VEL
LIN {X 0,Y 641.598,Z 935.412,A -85,B 0,C 180,E1 28678.528,E2 28678.528} C_VEL
LIN {X 0,Y 658.096,Z 910.47,A -85,B 0,C 180,E1 28677.874,E2 28677.874} C_VEL
LIN {X 0,Y 662.977,Z 903.074,A -85,B 0,C 180,E1 28677.689,E2 28677.689} C_VEL
LIN {X 0,Y 651.696,Z 894.954,A -85,B 0,C 180,E1 28676.74,E2 28676.74} C_VEL
LIN {X 0,Y 641.454,Z 885.193,A -85,B 0,C 180,E1 28675.706,E2 28675.706} C_VEL
LIN {X 0,Y 632.715,Z 874.063,A -85,B 0,C 180,E1 28674.632,E2 28674.632} C_VEL
LIN {X 0,Y 625.414,Z 861.409,A -85,B 0,C 180,E1 28673.505,E2 28673.505} C_VEL
LIN {X 0,Y 619.514,Z 846.572,A -85,B 0,C 180,E1 28672.286,E2 28672.286} C_VEL
LIN {X 0,Y 615.496,Z 830.19,A -85,B 0,C 180,E1 28671.046,E2 28671.046} C_VEL
LIN {X 0,Y 613.437,Z 813.302,A -85,B 0,C 180,E1 28669.859,E2 28669.859} C_VEL
LIN {X 0,Y 612.985,Z 791.643,A -85,B 0,C 180,E1 28668.442,E2 28668.442} C_VEL
LIN {X 0,Y 617.059,Z 730.126,A -85,B 0,C 180,E1 28664.653,E2 28664.653} C_VEL
LIN {X 0,Y 618.247,Z 714.472,A -85,B 0,C 180,E1 28663.677,E2 28663.677} C_VEL
LIN {X 0,Y 606.879,Z 688.829,A -85,B 0,C 180,E1 28660.976,E2 28660.976} C_VEL
LIN {X 0,Y 596.62,Z 666.622,A -85,B 0,C 180,E1 28658.446,E2 28658.446} C_VEL
LIN {X 0,Y 595.959,Z 665.352,A -85,B 0,C 180,E1 28658.26,E2 28658.26} C_VEL
LIN {X 0,Y 598.07,Z 668.996,A -85,B 0,C 180,E1 28657.606,E2 28657.606} C_VEL
LIN {X 0,Y 602.161,Z 678.41,A -85,B 0,C 180,E1 28656.195,E2 28656.195} C_VEL
LIN {X 0,Y 606.414,Z 691.139,A -85,B 0,C 180,E1 28654.556,E2 28654.556} C_VEL
LIN {X 0,Y 608.927,Z 701.376,A -85,B 0,C 180,E1 28653.373,E2 28653.373} C_VEL
LIN {X 0,Y 608.611,Z 709.812,A -85,B 0,C 180,E1 28652.67,E2 28652.67} C_VEL
LIN {X 0,Y 612.497,Z 728.046,A -85,B 0,C 180,E1 28651.974,E2 28651.974} C_VEL
LIN {X 0,Y 613.053,Z 732.448,A -85,B 0,C 180,E1 28651.846,E2 28651.846} C_VEL
LIN {X 0,Y 608.983,Z 839.422,A -85,B 0,C 180,E1 28650.125,E2 28650.125} C_VEL
LIN {X 0,Y 606.244,Z 946.949,A -85,B 0,C 180,E1 28648.539,E2 28648.539} C_VEL
LIN {X 0,Y 605.02,Z 1010.911,A -85,B 0,C 180,E1 28647.636,E2 28647.636} C_VEL
LIN {X 0,Y 604.315,Z 1033.288,A -85,B 0,C 180,E1 28647.149,E2 28647.149} C_VEL
LIN {X 0,Y 603.401,Z 1055.967,A -85,B 0,C 180,E1 28646.472,E2 28646.472} C_VEL
LIN {X 0,Y 602.355,Z 1077.115,A -85,B 0,C 180,E1 28645.661,E2 28645.661} C_VEL
LIN {X 0,Y 601.225,Z 1096.927,A -85,B 0,C 180,E1 28644.725,E2 28644.725} C_VEL
LIN {X 0,Y 599.976,Z 1116.107,A -85,B 0,C 180,E1 28643.629,E2 28643.629} C_VEL
LIN {X 0,Y 598.66,Z 1135.194,A -85,B 0,C 180,E1 28642.332,E2 28642.332} C_VEL
LIN {X 0,Y 597.398,Z 1152.602,A -85,B 0,C 180,E1 28640.94,E2 28640.94} C_VEL
LIN {X 0,Y 596.223,Z 1168.543,A -85,B 0,C 180,E1 28639.445,E2 28639.445} C_VEL
LIN {X 0,Y 595.196,Z 1182.564,A -85,B 0,C 180,E1 28637.904,E2 28637.904} C_VEL
LIN {X 0,Y 594.203,Z 1196.731,A -85,B 0,C 180,E1 28636.085,E2 28636.085} C_VEL
LIN {X 0,Y 593.472,Z 1208.297,A -85,B 0,C 180,E1 28634.34,E2 28634.34} C_VEL
LIN {X 0,Y 592.867,Z 1218.736,A -85,B 0,C 180,E1 28632.443,E2 28632.443} C_VEL
LIN {X 0,Y 592.458,Z 1227.589,A -85,B 0,C 180,E1 28630.502,E2 28630.502} C_VEL
LIN {X 0,Y 592.182,Z 1234.848,A -85,B 0,C 180,E1 28628.545,E2 28628.545} C_VEL
LIN {X 0,Y 592.035,Z 1240.619,A -85,B 0,C 180,E1 28626.497,E2 28626.497} C_VEL
LIN {X 0,Y 591.958,Z 1244.907,A -85,B 0,C 180,E1 28624.359,E2 28624.359} C_VEL
LIN {X 0,Y 591.926,Z 1247.457,A -85,B 0,C 180,E1 28622.323,E2 28622.323} C_VEL
LIN {X 0,Y 591.927,Z 1248.412,A -85,B 0,C 180,E1 28620.29,E2 28620.29} C_VEL
LIN {X 0,Y 591.934,Z 1247.809,A -85,B 0,C 180,E1 28618.161,E2 28618.161} C_VEL
LIN {X 0,Y 591.94,Z 1245.754,A -85,B 0,C 180,E1 28616.126,E2 28616.126} C_VEL
LIN {X 0,Y 591.991,Z 1242.04,A -85,B 0,C 180,E1 28614.086,E2 28614.086} C_VEL
LIN {X 0,Y 592.121,Z 1236.44,A -85,B 0,C 180,E1 28611.943,E2 28611.943} C_VEL
LIN {X 0,Y 592.359,Z 1229.354,A -85,B 0,C 180,E1 28609.889,E2 28609.889} C_VEL
LIN {X 0,Y 592.741,Z 1220.803,A -85,B 0,C 180,E1 28607.926,E2 28607.926} C_VEL
LIN {X 0,Y 593.279,Z 1210.88,A -85,B 0,C 180,E1 28606.054,E2 28606.054} C_VEL
LIN {X 0,Y 594.026,Z 1199.071,A -85,B 0,C 180,E1 28604.176,E2 28604.176} C_VEL
LIN {X 0,Y 594.962,Z 1185.819,A -85,B 0,C 180,E1 28602.392,E2 28602.392} C_VEL
LIN {X 0,Y 596.064,Z 1170.977,A -85,B 0,C 180,E1 28600.703,E2 28600.703} C_VEL
LIN {X 0,Y 597.341,Z 1154.632,A -85,B 0,C 180,E1 28599.112,E2 28599.112} C_VEL
LIN {X 0,Y 598.686,Z 1137.297,A -85,B 0,C 180,E1 28597.669,E2 28597.669} C_VEL
LIN {X 0,Y 600.074,Z 1119.061,A -85,B 0,C 180,E1 28596.375,E2 28596.375} C_VEL
LIN {X 0,Y 601.423,Z 1099.798,A -85,B 0,C 180,E1 28595.231,E2 28595.231} C_VEL
LIN {X 0,Y 602.717,Z 1079.795,A -85,B 0,C 180,E1 28594.237,E2 28594.237} C_VEL
LIN {X 0,Y 603.902,Z 1059.08,A -85,B 0,C 180,E1 28593.392,E2 28593.392} C_VEL
LIN {X 0,Y 604.945,Z 1037.425,A -85,B 0,C 180,E1 28592.699,E2 28592.699} C_VEL
LIN {X 0,Y 605.732,Z 1015.446,A -85,B 0,C 180,E1 28592.176,E2 28592.176} C_VEL
LIN {X 0,Y 606.392,Z 989.072,A -85,B 0,C 180,E1 28591.757,E2 28591.757} C_VEL
LIN {X 0,Y 610.43,Z 773.93,A -85,B 0,C 180,E1 28588.879,E2 28588.879} C_VEL
LIN {X 0,Y 611.197,Z 730.031,A -85,B 0,C 180,E1 28588.266,E2 28588.266} C_VEL
LIN {X 0,Y 605.137,Z 702.858,A -85,B 0,C 180,E1 28587.491,E2 28587.491} C_VEL
LIN {X 0,Y 605.251,Z 696.089,A -85,B 0,C 180,E1 28586.886,E2 28586.886} C_VEL
LIN {X 0,Y 602.1,Z 685.7,A -85,B 0,C 180,E1 28585.744,E2 28585.744} C_VEL
LIN {X 0,Y 599.752,Z 681.222,A -85,B 0,C 180,E1 28585.183,E2 28585.183} C_VEL
LIN {X 0,Y 589.555,Z 670.726,A -85,B 0,C 180,E1 28583.548,E2 28583.548} C_VEL
LIN {X 0,Y 587.812,Z 667.527,A -85,B 0,C 180,E1 28583.136,E2 28583.136} C_VEL
LIN {X 0,Y 585.252,Z 659.765,A -85,B 0,C 180,E1 28582.23,E2 28582.23} C_VEL
LIN {X 0,Y 585.263,Z 659.764,A -85,B 0,C 180,E1 28578.871,E2 28578.871} C_VEL
LIN {X 0,Y 585.258,Z 659.768,A -85,B 0,C 180,E1 28575.535,E2 28575.535} C_VEL
LIN {X 0,Y 585.244,Z 659.763,A -85,B 0,C 180,E1 28572.287,E2 28572.287} C_VEL
LIN {X 0,Y 585.243,Z 659.769,A -85,B 0,C 180,E1 28569.083,E2 28569.083} C_VEL
LIN {X 0,Y 585.258,Z 659.769,A -85,B 0,C 180,E1 28565.875,E2 28565.875} C_VEL
LIN {X 0,Y 585.262,Z 659.769,A -85,B 0,C 180,E1 28562.559,E2 28562.559} C_VEL
LIN {X 0,Y 585.249,Z 659.765,A -85,B 0,C 180,E1 28559.364,E2 28559.364} C_VEL
LIN {X 0,Y 585.254,Z 659.764,A -85,B 0,C 180,E1 28556.017,E2 28556.017} C_VEL
LIN {X 0,Y 585.252,Z 659.764,A -85,B 0,C 180,E1 28552.693,E2 28552.693} C_VEL
LIN {X 0,Y 585.245,Z 659.763,A -85,B 0,C 180,E1 28549.422,E2 28549.422} C_VEL
LIN {X 0,Y 585.242,Z 659.768,A -85,B 0,C 180,E1 28546.171,E2 28546.171} C_VEL
LIN {X 0,Y 585.256,Z 659.761,A -85,B 0,C 180,E1 28542.934,E2 28542.934} C_VEL
LIN {X 0,Y 585.247,Z 659.768,A -85,B 0,C 180,E1 28539.64,E2 28539.64} C_VEL
LIN {X 0,Y 585.255,Z 659.764,A -85,B 0,C 180,E1 28536.377,E2 28536.377} C_VEL
LIN {X 0,Y 585.251,Z 659.761,A -85,B 0,C 180,E1 28533.037,E2 28533.037} C_VEL
LIN {X 0,Y 585.246,Z 659.759,A -85,B 0,C 180,E1 28529.708,E2 28529.708} C_VEL
LIN {X 0,Y 585.242,Z 659.761,A -85,B 0,C 180,E1 28526.475,E2 28526.475} C_VEL
LIN {X 0,Y 585.246,Z 659.766,A -85,B 0,C 180,E1 28523.231,E2 28523.231} C_VEL
LIN {X 0,Y 585.245,Z 659.769,A -85,B 0,C 180,E1 28520.065,E2 28520.065} C_VEL
LIN {X 0,Y 585.247,Z 659.766,A -85,B 0,C 180,E1 28516.767,E2 28516.767} C_VEL
LIN {X 0,Y 585.251,Z 659.764,A -85,B 0,C 180,E1 28513.526,E2 28513.526} C_VEL
LIN {X 0,Y 585.255,Z 659.761,A -85,B 0,C 180,E1 28510.126,E2 28510.126} C_VEL
LIN {X 0,Y 585.247,Z 659.767,A -85,B 0,C 180,E1 28506.806,E2 28506.806} C_VEL
LIN {X 0,Y 585.257,Z 659.767,A -85,B 0,C 180,E1 28503.539,E2 28503.539} C_VEL
LIN {X 0,Y 585.261,Z 659.766,A -85,B 0,C 180,E1 28500.215,E2 28500.215} C_VEL
LIN {X 0,Y 585.248,Z 659.757,A -85,B 0,C 180,E1 28496.977,E2 28496.977} C_VEL
LIN {X 0,Y 585.253,Z 659.758,A -85,B 0,C 180,E1 28493.644,E2 28493.644} C_VEL
LIN {X 0,Y 585.254,Z 659.764,A -85,B 0,C 180,E1 28490.288,E2 28490.288} C_VEL
LIN {X 0,Y 585.245,Z 659.771,A -85,B 0,C 180,E1 28486.991,E2 28486.991} C_VEL
LIN {X 0,Y 585.269,Z 659.96,A -85,B 0,C 180,E1 28486.805,E2 28486.805} C_VEL
LIN {X 0,Y 594.903,Z 686.068,A -85,B 0,C 180,E1 28483.862,E2 28483.862} C_VEL
LIN {X 0,Y 600.998,Z 703.898,A -85,B 0,C 180,E1 28481.957,E2 28481.957} C_VEL
LIN {X 0,Y 598.78,Z 741.482,A -85,B 0,C 180,E1 28479.017,E2 28479.017} C_VEL
LIN {X 0,Y 596.322,Z 783.986,A -85,B 0,C 180,E1 28475.756,E2 28475.756} C_VEL
LIN {X 0,Y 594.057,Z 827.304,A -85,B 0,C 180,E1 28472.475,E2 28472.475} C_VEL
LIN {X 0,Y 591.884,Z 873.668,A -85,B 0,C 180,E1 28469.002,E2 28469.002} C_VEL
LIN {X 0,Y 590.818,Z 901.628,A -85,B 0,C 180,E1 28466.961,E2 28466.961} C_VEL
LIN {X 0,Y 591.646,Z 910.285,A -85,B 0,C 180,E1 28466.793,E2 28466.793} C_VEL
LIN {X 0,Y 589.087,Z 1046.153,A -85,B 0,C 180,E1 28464.68,E2 28464.68} C_VEL
LIN {X 0,Y 588.792,Z 1062.922,A -85,B 0,C 180,E1 28464.231,E2 28464.231} C_VEL
LIN {X 0,Y 588.376,Z 1078.21,A -85,B 0,C 180,E1 28463.645,E2 28463.645} C_VEL
LIN {X 0,Y 587.801,Z 1094.17,A -85,B 0,C 180,E1 28462.821,E2 28462.821} C_VEL
LIN {X 0,Y 587.233,Z 1108.099,A -85,B 0,C 180,E1 28461.894,E2 28461.894} C_VEL
LIN {X 0,Y 586.625,Z 1121.604,A -85,B 0,C 180,E1 28460.765,E2 28460.765} C_VEL
LIN {X 0,Y 586.119,Z 1132.466,A -85,B 0,C 180,E1 28459.638,E2 28459.638} C_VEL
LIN {X 0,Y 585.622,Z 1142.788,A -85,B 0,C 180,E1 28458.31,E2 28458.31} C_VEL
LIN {X 0,Y 585.232,Z 1151.6,A -85,B 0,C 180,E1 28456.885,E2 28456.885} C_VEL
LIN {X 0,Y 584.939,Z 1158.796,A -85,B 0,C 180,E1 28455.364,E2 28455.364} C_VEL
LIN {X 0,Y 584.767,Z 1164.259,A -85,B 0,C 180,E1 28453.789,E2 28453.789} C_VEL
LIN {X 0,Y 584.676,Z 1167.956,A -85,B 0,C 180,E1 28452.143,E2 28452.143} C_VEL
LIN {X 0,Y 584.656,Z 1169.785,A -85,B 0,C 180,E1 28450.544,E2 28450.544} C_VEL
LIN {X 0,Y 584.71,Z 1169.781,A -85,B 0,C 180,E1 28448.853,E2 28448.853} C_VEL
LIN {X 0,Y 584.821,Z 1168.073,A -85,B 0,C 180,E1 28447.269,E2 28447.269} C_VEL
LIN {X 0,Y 585.022,Z 1164.3,A -85,B 0,C 180,E1 28445.591,E2 28445.591} C_VEL
LIN {X 0,Y 585.324,Z 1159.3,A -85,B 0,C 180,E1 28444.114,E2 28444.114} C_VEL
LIN {X 0,Y 585.765,Z 1151.922,A -85,B 0,C 180,E1 28442.544,E2 28442.544} C_VEL
LIN {X 0,Y 586.303,Z 1143.596,A -85,B 0,C 180,E1 28441.173,E2 28441.173} C_VEL
LIN {X 0,Y 586.977,Z 1132.99,A -85,B 0,C 180,E1 28439.805,E2 28439.805} C_VEL
LIN {X 0,Y 587.668,Z 1121.712,A -85,B 0,C 180,E1 28438.635,E2 28438.635} C_VEL
LIN {X 0,Y 588.421,Z 1108.208,A -85,B 0,C 180,E1 28437.516,E2 28437.516} C_VEL
LIN {X 0,Y 589.079,Z 1095.019,A -85,B 0,C 180,E1 28436.643,E2 28436.643} C_VEL
LIN {X 0,Y 589.712,Z 1079.918,A -85,B 0,C 180,E1 28435.868,E2 28435.868} C_VEL
LIN {X 0,Y 590.183,Z 1064.612,A -85,B 0,C 180,E1 28435.275,E2 28435.275} C_VEL
LIN {X 0,Y 590.477,Z 1047.652,A -85,B 0,C 180,E1 28434.827,E2 28434.827} C_VEL
LIN {X 0,Y 595.561,Z 911.683,A -85,B 0,C 180,E1 28432.233,E2 28432.233} C_VEL
LIN {X 0,Y 599.314,Z 865.899,A -85,B 0,C 180,E1 28428.548,E2 28428.548} C_VEL
LIN {X 0,Y 603.616,Z 823.406,A -85,B 0,C 180,E1 28425.024,E2 28425.024} C_VEL
LIN {X 0,Y 608.674,Z 783.623,A -85,B 0,C 180,E1 28421.615,E2 28421.615} C_VEL
LIN {X 0,Y 614.209,Z 748.199,A -85,B 0,C 180,E1 28418.463,E2 28418.463} C_VEL
LIN {X 0,Y 617.521,Z 727.844,A -85,B 0,C 180,E1 28416.526,E2 28416.526} C_VEL
LIN {X 0,Y 614.168,Z 717.252,A -85,B 0,C 180,E1 28414.625,E2 28414.625} C_VEL
LIN {X 0,Y 610.957,Z 708.119,A -85,B 0,C 180,E1 28412.62,E2 28412.62} C_VEL
LIN {X 0,Y 608.921,Z 703.242,A -85,B 0,C 180,E1 28411.241,E2 28411.241} C_VEL
LIN {X 0,Y 607.824,Z 700.346,A -85,B 0,C 180,E1 28410.289,E2 28410.289} C_VEL
LIN {X 0,Y 606.655,Z 697.009,A -85,B 0,C 180,E1 28408.943,E2 28408.943} C_VEL
LIN {X 0,Y 605.475,Z 694.242,A -85,B 0,C 180,E1 28406.977,E2 28406.977} C_VEL
LIN {X 0,Y 605.561,Z 693.306,A -85,B 0,C 180,E1 28405.813,E2 28405.813} C_VEL
LIN {X 0,Y 605.828,Z 693.762,A -85,B 0,C 180,E1 28404.365,E2 28404.365} C_VEL
LIN {X 0,Y 607.037,Z 696.989,A -85,B 0,C 180,E1 28402.331,E2 28402.331} C_VEL
LIN {X 0,Y 607.902,Z 698.368,A -85,B 0,C 180,E1 28401.676,E2 28401.676} C_VEL
LIN {X 0,Y 609.854,Z 702.875,A -85,B 0,C 180,E1 28400.251,E2 28400.251} C_VEL
LIN {X 0,Y 612.421,Z 708.848,A -85,B 0,C 180,E1 28398.819,E2 28398.819} C_VEL
LIN {X 0,Y 615.61,Z 717.632,A -85,B 0,C 180,E1 28397.24,E2 28397.24} C_VEL
LIN {X 0,Y 616.373,Z 720.339,A -85,B 0,C 180,E1 28396.846,E2 28396.846} C_VEL
LIN {X 0,Y 609.975,Z 755.055,A -85,B 0,C 180,E1 28394.355,E2 28394.355} C_VEL
LIN {X 0,Y 605.527,Z 789.793,A -85,B 0,C 180,E1 28391.969,E2 28391.969} C_VEL
LIN {X 0,Y 604.897,Z 810.948,A -85,B 0,C 180,E1 28390.449,E2 28390.449} C_VEL
LIN {X 0,Y 606.263,Z 828.652,A -85,B 0,C 180,E1 28389.106,E2 28389.106} C_VEL
LIN {X 0,Y 609.7,Z 845.219,A -85,B 0,C 180,E1 28387.77,E2 28387.77} C_VEL
LIN {X 0,Y 615.034,Z 859.97,A -85,B 0,C 180,E1 28386.512,E2 28386.512} C_VEL
LIN {X 0,Y 621.779,Z 872.708,A -85,B 0,C 180,E1 28385.372,E2 28385.372} C_VEL
LIN {X 0,Y 630.996,Z 885.299,A -85,B 0,C 180,E1 28384.19,E2 28384.19} C_VEL
LIN {X 0,Y 642.06,Z 896.455,A -85,B 0,C 180,E1 28383.087,E2 28383.087} C_VEL
LIN {X 0,Y 651.777,Z 904.277,A -85,B 0,C 180,E1 28382.288,E2 28382.288} C_VEL
LIN {X 0,Y 634.602,Z 929.715,A -85,B 0,C 180,E1 28381.592,E2 28381.592} C_VEL
LIN {X 0,Y 623.532,Z 948.874,A -85,B 0,C 180,E1 28380.979,E2 28380.979} C_VEL
LIN {X 0,Y 615.489,Z 966.044,A -85,B 0,C 180,E1 28380.345,E2 28380.345} C_VEL
LIN {X 0,Y 611.655,Z 974.681,A -85,B 0,C 180,E1 28380.013,E2 28380.013} C_VEL
LIN {X 0,Y 605.061,Z 990.301,A -85,B 0,C 180,E1 28379.392,E2 28379.392} C_VEL
LIN {X 0,Y 600.243,Z 1005.069,A -85,B 0,C 180,E1 28378.768,E2 28378.768} C_VEL
LIN {X 0,Y 598.289,Z 1026.585,A -85,B 0,C 180,E1 28378.555,E2 28378.555} C_VEL
LIN {X 0,Y 597.513,Z 1064.146,A -85,B 0,C 180,E1 28378.015,E2 28378.015} C_VEL
LIN {X 0,Y 596.686,Z 1085.659,A -85,B 0,C 180,E1 28377.543,E2 28377.543} C_VEL
LIN {X 0,Y 595.624,Z 1107.152,A -85,B 0,C 180,E1 28376.897,E2 28376.897} C_VEL
LIN {X 0,Y 594.351,Z 1129.258,A -85,B 0,C 180,E1 28376.044,E2 28376.044} C_VEL
LIN {X 0,Y 593.061,Z 1149.351,A -85,B 0,C 180,E1 28375.087,E2 28375.087} C_VEL
LIN {X 0,Y 591.728,Z 1168.605,A -85,B 0,C 180,E1 28373.976,E2 28373.976} C_VEL
LIN {X 0,Y 590.349,Z 1187.124,A -85,B 0,C 180,E1 28372.715,E2 28372.715} C_VEL
LIN {X 0,Y 589.061,Z 1204.873,A -85,B 0,C 180,E1 28371.298,E2 28371.298} C_VEL
LIN {X 0,Y 587.837,Z 1221.547,A -85,B 0,C 180,E1 28369.743,E2 28369.743} C_VEL
LIN {X 0,Y 586.753,Z 1236.816,A -85,B 0,C 180,E1 28368.066,E2 28368.066} C_VEL
LIN {X 0,Y 585.857,Z 1250.949,A -85,B 0,C 180,E1 28366.253,E2 28366.253} C_VEL
LIN {X 0,Y 585.177,Z 1262.983,A -85,B 0,C 180,E1 28364.445,E2 28364.445} C_VEL
LIN {X 0,Y 584.692,Z 1273.627,A -85,B 0,C 180,E1 28362.542,E2 28362.542} C_VEL
LIN {X 0,Y 584.338,Z 1282.85,A -85,B 0,C 180,E1 28360.548,E2 28360.548} C_VEL
LIN {X 0,Y 584.172,Z 1290.279,A -85,B 0,C 180,E1 28358.562,E2 28358.562} C_VEL
LIN {X 0,Y 584.08,Z 1295.756,A -85,B 0,C 180,E1 28356.683,E2 28356.683} C_VEL
LIN {X 0,Y 584.065,Z 1300.813,A -85,B 0,C 180,E1 28354.319,E2 28354.319} C_VEL
LIN {X 0,Y 584.059,Z 1303.175,A -85,B 0,C 180,E1 28352.55,E2 28352.55} C_VEL
LIN {X 0,Y 584.066,Z 1304.301,A -85,B 0,C 180,E1 28350.881,E2 28350.881} C_VEL
LIN {X 0,Y 584.059,Z 1304.362,A -85,B 0,C 180,E1 28349.214,E2 28349.214} C_VEL
LIN {X 0,Y 584.048,Z 1303.271,A -85,B 0,C 180,E1 28347.448,E2 28347.448} C_VEL
LIN {X 0,Y 584.04,Z 1300.535,A -85,B 0,C 180,E1 28345.383,E2 28345.383} C_VEL
LIN {X 0,Y 584.063,Z 1295.967,A -85,B 0,C 180,E1 28343.314,E2 28343.314} C_VEL
LIN {X 0,Y 584.161,Z 1290.348,A -85,B 0,C 180,E1 28341.435,E2 28341.435} C_VEL
LIN {X 0,Y 584.328,Z 1282.828,A -85,B 0,C 180,E1 28339.449,E2 28339.449} C_VEL
LIN {X 0,Y 584.675,Z 1273.375,A -85,B 0,C 180,E1 28337.455,E2 28337.455} C_VEL
LIN {X 0,Y 585.153,Z 1262.512,A -85,B 0,C 180,E1 28335.552,E2 28335.552} C_VEL
LIN {X 0,Y 585.85,Z 1249.545,A -85,B 0,C 180,E1 28333.643,E2 28333.643} C_VEL
LIN {X 0,Y 586.638,Z 1236.437,A -85,B 0,C 180,E1 28332.005,E2 28332.005} C_VEL
LIN {X 0,Y 587.468,Z 1223.746,A -85,B 0,C 180,E1 28330.615,E2 28330.615} C_VEL
LIN {X 0,Y 588.566,Z 1207.967,A -85,B 0,C 180,E1 28329.098,E2 28329.098} C_VEL
LIN {X 0,Y 589.835,Z 1189.922,A -85,B 0,C 180,E1 28327.63,E2 28327.63} C_VEL
LIN {X 0,Y 591.108,Z 1171.937,A -85,B 0,C 180,E1 28326.365,E2 28326.365} C_VEL
LIN {X 0,Y 592.424,Z 1152.219,A -85,B 0,C 180,E1 28325.201,E2 28325.201} C_VEL
LIN {X 0,Y 593.804,Z 1130.737,A -85,B 0,C 180,E1 28324.142,E2 28324.142} C_VEL
LIN {X 0,Y 595.03,Z 1110.29,A -85,B 0,C 180,E1 28323.314,E2 28323.314} C_VEL
LIN {X 0,Y 596.125,Z 1088.181,A -85,B 0,C 180,E1 28322.616,E2 28322.616} C_VEL
LIN {X 0,Y 597.11,Z 1065.3,A -85,B 0,C 180,E1 28322.079,E2 28322.079} C_VEL
LIN {X 0,Y 597.743,Z 1041.947,A -85,B 0,C 180,E1 28321.702,E2 28321.702} C_VEL
LIN {X 0,Y 598.443,Z 1018.74,A -85,B 0,C 180,E1 28321.409,E2 28321.409} C_VEL
LIN {X 0,Y 598.761,Z 1016.325,A -85,B 0,C 180,E1 28321.361,E2 28321.361} C_VEL
LIN {X 0,Y 605.023,Z 996.344,A -85,B 0,C 180,E1 28320.453,E2 28320.453} C_VEL
LIN {X 0,Y 611.29,Z 980.594,A -85,B 0,C 180,E1 28319.802,E2 28319.802} C_VEL
LIN {X 0,Y 616.408,Z 969.521,A -85,B 0,C 180,E1 28319.379,E2 28319.379} C_VEL
LIN {X 0,Y 623.894,Z 953.276,A -85,B 0,C 180,E1 28318.77,E2 28318.77} C_VEL
LIN {X 0,Y 634.842,Z 933.934,A -85,B 0,C 180,E1 28318.154,E2 28318.154} C_VEL
LIN {X 0,Y 650.753,Z 909.821,A -85,B 0,C 180,E1 28317.517,E2 28317.517} C_VEL
LIN {X 0,Y 653.188,Z 906.023,A -85,B 0,C 180,E1 28317.416,E2 28317.416} C_VEL
LIN {X 0,Y 642.122,Z 897.159,A -85,B 0,C 180,E1 28316.417,E2 28316.417} C_VEL
LIN {X 0,Y 632.144,Z 886.67,A -85,B 0,C 180,E1 28315.337,E2 28315.337} C_VEL
LIN {X 0,Y 623.377,Z 874.255,A -85,B 0,C 180,E1 28314.164,E2 28314.164} C_VEL
LIN {X 0,Y 616.666,Z 861.119,A -85,B 0,C 180,E1 28313.018,E2 28313.018} C_VEL
LIN {X 0,Y 611.464,Z 846.362,A -85,B 0,C 180,E1 28311.82,E2 28311.82} C_VEL
LIN {X 0,Y 607.895,Z 829.682,A -85,B 0,C 180,E1 28310.564,E2 28310.564} C_VEL
LIN {X 0,Y 606.167,Z 811.253,A -85,B 0,C 180,E1 28309.277,E2 28309.277} C_VEL
LIN {X 0,Y 606.207,Z 789.061,A -85,B 0,C 180,E1 28307.831,E2 28307.831} C_VEL
LIN {X 0,Y 610.207,Z 733.821,A -85,B 0,C 180,E1 28304.402,E2 28304.402} C_VEL
LIN {X 0,Y 611.378,Z 717.81,A -85,B 0,C 180,E1 28303.385,E2 28303.385} C_VEL
LIN {X 0,Y 599.704,Z 691.358,A -85,B 0,C 180,E1 28300.561,E2 28300.561} C_VEL
LIN {X 0,Y 590.823,Z 671.961,A -85,B 0,C 180,E1 28298.313,E2 28298.313} C_VEL
LIN {X 0,Y 591.81,Z 672.931,A -85,B 0,C 180,E1 28298.063,E2 28298.063} C_VEL
LIN {X 0,Y 595.496,Z 681.37,A -85,B 0,C 180,E1 28296.71,E2 28296.71} C_VEL
LIN {X 0,Y 599.446,Z 692.848,A -85,B 0,C 180,E1 28295.133,E2 28295.133} C_VEL
LIN {X 0,Y 602.461,Z 705.039,A -85,B 0,C 180,E1 28293.665,E2 28293.665} C_VEL
LIN {X 0,Y 602.291,Z 710.786,A -85,B 0,C 180,E1 28293.194,E2 28293.194} C_VEL
LIN {X 0,Y 606.037,Z 728.578,A -85,B 0,C 180,E1 28292.471,E2 28292.471} C_VEL
LIN {X 0,Y 606.756,Z 733.986,A -85,B 0,C 180,E1 28292.295,E2 28292.295} C_VEL
LIN {X 0,Y 602.23,Z 840.056,A -85,B 0,C 180,E1 28290.527,E2 28290.527} C_VEL
LIN {X 0,Y 599.225,Z 944.478,A -85,B 0,C 180,E1 28288.932,E2 28288.932} C_VEL
LIN {X 0,Y 597.775,Z 1011.924,A -85,B 0,C 180,E1 28287.95,E2 28287.95} C_VEL
LIN {X 0,Y 597.019,Z 1034.348,A -85,B 0,C 180,E1 28287.448,E2 28287.448} C_VEL
LIN {X 0,Y 596.061,Z 1056.602,A -85,B 0,C 180,E1 28286.77,E2 28286.77} C_VEL
LIN {X 0,Y 594.967,Z 1077.5,A -85,B 0,C 180,E1 28285.958,E2 28285.958} C_VEL
LIN {X 0,Y 593.767,Z 1097.422,A -85,B 0,C 180,E1 28285.004,E2 28285.004} C_VEL
LIN {X 0,Y 592.455,Z 1116.582,A -85,B 0,C 180,E1 28283.894,E2 28283.894} C_VEL
LIN {X 0,Y 591.067,Z 1135.649,A -85,B 0,C 180,E1 28282.582,E2 28282.582} C_VEL
LIN {X 0,Y 589.777,Z 1152.534,A -85,B 0,C 180,E1 28281.221,E2 28281.221} C_VEL
LIN {X 0,Y 588.573,Z 1168.06,A -85,B 0,C 180,E1 28279.752,E2 28279.752} C_VEL
LIN {X 0,Y 587.445,Z 1182.598,A -85,B 0,C 180,E1 28278.149,E2 28278.149} C_VEL
LIN {X 0,Y 586.46,Z 1195.904,A -85,B 0,C 180,E1 28276.441,E2 28276.441} C_VEL
LIN {X 0,Y 585.646,Z 1207.845,A -85,B 0,C 180,E1 28274.637,E2 28274.637} C_VEL
LIN {X 0,Y 584.997,Z 1218.337,A -85,B 0,C 180,E1 28272.738,E2 28272.738} C_VEL
LIN {X 0,Y 584.516,Z 1227.875,A -85,B 0,C 180,E1 28270.646,E2 28270.646} C_VEL
LIN {X 0,Y 584.221,Z 1235.182,A -85,B 0,C 180,E1 28268.662,E2 28268.662} C_VEL
LIN {X 0,Y 584.056,Z 1240.974,A -85,B 0,C 180,E1 28266.586,E2 28266.586} C_VEL
LIN {X 0,Y 583.974,Z 1245.283,A -85,B 0,C 180,E1 28264.419,E2 28264.419} C_VEL
LIN {X 0,Y 583.938,Z 1247.841,A -85,B 0,C 180,E1 28262.355,E2 28262.355} C_VEL
LIN {X 0,Y 583.936,Z 1248.791,A -85,B 0,C 180,E1 28260.294,E2 28260.294} C_VEL
LIN {X 0,Y 583.943,Z 1248.177,A -85,B 0,C 180,E1 28258.136,E2 28258.136} C_VEL
LIN {X 0,Y 583.951,Z 1246.099,A -85,B 0,C 180,E1 28256.073,E2 28256.073} C_VEL
LIN {X 0,Y 584.008,Z 1242.358,A -85,B 0,C 180,E1 28254.005,E2 28254.005} C_VEL
LIN {X 0,Y 584.153,Z 1236.718,A -85,B 0,C 180,E1 28251.832,E2 28251.832} C_VEL
LIN {X 0,Y 584.411,Z 1229.589,A -85,B 0,C 180,E1 28249.75,E2 28249.75} C_VEL
LIN {X 0,Y 584.818,Z 1221.003,A -85,B 0,C 180,E1 28247.76,E2 28247.76} C_VEL
LIN {X 0,Y 585.399,Z 1211.023,A -85,B 0,C 180,E1 28245.862,E2 28245.862} C_VEL
LIN {X 0,Y 586.196,Z 1199.144,A -85,B 0,C 180,E1 28243.959,E2 28243.959} C_VEL
LIN {X 0,Y 587.196,Z 1185.834,A -85,B 0,C 180,E1 28242.151,E2 28242.151} C_VEL
LIN {X 0,Y 588.364,Z 1170.915,A -85,B 0,C 180,E1 28240.44,E2 28240.44} C_VEL
LIN {X 0,Y 589.623,Z 1155.583,A -85,B 0,C 180,E1 28238.93,E2 28238.93} C_VEL
LIN {X 0,Y 591.023,Z 1138.452,A -85,B 0,C 180,E1 28237.477,E2 28237.477} C_VEL
LIN {X 0,Y 592.465,Z 1120.262,A -85,B 0,C 180,E1 28236.167,E2 28236.167} C_VEL
LIN {X 0,Y 593.884,Z 1101.044,A -85,B 0,C 180,E1 28235.001,E2 28235.001} C_VEL
LIN {X 0,Y 595.307,Z 1080.169,A -85,B 0,C 180,E1 28233.946,E2 28233.946} C_VEL
LIN {X 0,Y 596.559,Z 1059.344,A -85,B 0,C 180,E1 28233.086,E2 28233.086} C_VEL
LIN {X 0,Y 597.642,Z 1037.886,A -85,B 0,C 180,E1 28232.391,E2 28232.391} C_VEL
LIN {X 0,Y 598.465,Z 1016.082,A -85,B 0,C 180,E1 28231.863,E2 28231.863} C_VEL
LIN {X 0,Y 599.168,Z 989.663,A -85,B 0,C 180,E1 28231.434,E2 28231.434} C_VEL
LIN {X 0,Y 603.344,Z 780.995,A -85,B 0,C 180,E1 28228.597,E2 28228.597} C_VEL
LIN {X 0,Y 604.304,Z 731.505,A -85,B 0,C 180,E1 28227.894,E2 28227.894} C_VEL
LIN {X 0,Y 597.997,Z 703.116,A -85,B 0,C 180,E1 28227.075,E2 28227.075} C_VEL
LIN {X 0,Y 598.049,Z 699.16,A -85,B 0,C 180,E1 28226.717,E2 28226.717} C_VEL
LIN {X 0,Y 591.555,Z 678.413,A -85,B 0,C 180,E1 28224.393,E2 28224.393} C_VEL
LIN {X 0,Y 587.812,Z 667.527,A -85,B 0,C 180,E1 28223.136,E2 28223.136} C_VEL
LIN {X 0,Y 585.831,Z 664.664,A -85,B 0,C 180,E1 28222.732,E2 28222.732} C_VEL
LIN {X 0,Y 580.997,Z 661.925,A -85,B 0,C 180,E1 28222.089,E2 28222.089} C_VEL
LIN {X 0,Y 578.154,Z 660.981,A -85,B 0,C 180,E1 28221.56,E2 28221.56} C_VEL
LIN {X 0,Y 577.316,Z 660.757,A -85,B 0,C 180,E1 28221.121,E2 28221.121} C_VEL
LIN {X 0,Y 577.314,Z 660.756,A -85,B 0,C 180,E1 28217.694,E2 28217.694} C_VEL
LIN {X 0,Y 577.307,Z 660.757,A -85,B 0,C 180,E1 28214.406,E2 28214.406} C_VEL
LIN {X 0,Y 577.304,Z 660.76,A -85,B 0,C 180,E1 28211.112,E2 28211.112} C_VEL
LIN {X 0,Y 577.322,Z 660.754,A -85,B 0,C 180,E1 28207.816,E2 28207.816} C_VEL
LIN {X 0,Y 577.313,Z 660.754,A -85,B 0,C 180,E1 28204.47,E2 28204.47} C_VEL
LIN {X 0,Y 577.324,Z 660.752,A -85,B 0,C 180,E1 28201.176,E2 28201.176} C_VEL
LIN {X 0,Y 577.311,Z 660.752,A -85,B 0,C 180,E1 28197.882,E2 28197.882} C_VEL
LIN {X 0,Y 577.305,Z 660.754,A -85,B 0,C 180,E1 28194.563,E2 28194.563} C_VEL
LIN {X 0,Y 577.304,Z 660.755,A -85,B 0,C 180,E1 28191.33,E2 28191.33} C_VEL
LIN {X 0,Y 577.313,Z 660.757,A -85,B 0,C 180,E1 28188.062,E2 28188.062} C_VEL
LIN {X 0,Y 577.318,Z 660.757,A -85,B 0,C 180,E1 28184.751,E2 28184.751} C_VEL
LIN {X 0,Y 577.318,Z 660.753,A -85,B 0,C 180,E1 28181.389,E2 28181.389} C_VEL
LIN {X 0,Y 577.318,Z 660.746,A -85,B 0,C 180,E1 28177.966,E2 28177.966} C_VEL
LIN {X 0,Y 577.304,Z 660.751,A -85,B 0,C 180,E1 28174.77,E2 28174.77} C_VEL
LIN {X 0,Y 577.303,Z 660.754,A -85,B 0,C 180,E1 28171.49,E2 28171.49} C_VEL
LIN {X 0,Y 577.317,Z 660.755,A -85,B 0,C 180,E1 28168.314,E2 28168.314} C_VEL
LIN {X 0,Y 577.32,Z 660.756,A -85,B 0,C 180,E1 28164.934,E2 28164.934} C_VEL
LIN {X 0,Y 577.321,Z 660.752,A -85,B 0,C 180,E1 28161.636,E2 28161.636} C_VEL
LIN {X 0,Y 577.312,Z 660.75,A -85,B 0,C 180,E1 28158.31,E2 28158.31} C_VEL
LIN {X 0,Y 577.307,Z 660.752,A -85,B 0,C 180,E1 28155.046,E2 28155.046} C_VEL
LIN {X 0,Y 577.304,Z 660.755,A -85,B 0,C 180,E1 28151.836,E2 28151.836} C_VEL
LIN {X 0,Y 577.306,Z 660.756,A -85,B 0,C 180,E1 28148.567,E2 28148.567} C_VEL
LIN {X 0,Y 577.324,Z 660.753,A -85,B 0,C 180,E1 28145.332,E2 28145.332} C_VEL
LIN {X 0,Y 577.322,Z 660.755,A -85,B 0,C 180,E1 28142.009,E2 28142.009} C_VEL
LIN {X 0,Y 577.327,Z 660.752,A -85,B 0,C 180,E1 28138.698,E2 28138.698} C_VEL
LIN {X 0,Y 577.307,Z 660.76,A -85,B 0,C 180,E1 28135.356,E2 28135.356} C_VEL
LIN {X 0,Y 577.306,Z 660.76,A -85,B 0,C 180,E1 28132.061,E2 28132.061} C_VEL
LIN {X 0,Y 577.302,Z 660.753,A -85,B 0,C 180,E1 28128.843,E2 28128.843} C_VEL
LIN {X 0,Y 577.335,Z 660.889,A -85,B 0,C 180,E1 28127.332,E2 28127.332} C_VEL
LIN {X 0,Y 586.817,Z 686.534,A -85,B 0,C 180,E1 28124.376,E2 28124.376} C_VEL
LIN {X 0,Y 593.845,Z 706.915,A -85,B 0,C 180,E1 28122.176,E2 28122.176} C_VEL
LIN {X 0,Y 591.507,Z 744.434,A -85,B 0,C 180,E1 28119.214,E2 28119.214} C_VEL
LIN {X 0,Y 588.912,Z 786.949,A -85,B 0,C 180,E1 28115.919,E2 28115.919} C_VEL
LIN {X 0,Y 586.523,Z 830.408,A -85,B 0,C 180,E1 28112.596,E2 28112.596} C_VEL
LIN {X 0,Y 584.298,Z 876.326,A -85,B 0,C 180,E1 28109.134,E2 28109.134} C_VEL
LIN {X 0,Y 583.248,Z 902.244,A -85,B 0,C 180,E1 28107.222,E2 28107.222} C_VEL
LIN {X 0,Y 584.107,Z 911.169,A -85,B 0,C 180,E1 28107.046,E2 28107.046} C_VEL
LIN {X 0,Y 581.374,Z 1046.891,A -85,B 0,C 180,E1 28104.879,E2 28104.879} C_VEL
LIN {X 0,Y 581.069,Z 1063.431,A -85,B 0,C 180,E1 28104.429,E2 28104.429} C_VEL
LIN {X 0,Y 580.621,Z 1079.107,A -85,B 0,C 180,E1 28103.818,E2 28103.818} C_VEL
LIN {X 0,Y 580.032,Z 1094.72,A -85,B 0,C 180,E1 28103.001,E2 28103.001} C_VEL
LIN {X 0,Y 579.453,Z 1108.344,A -85,B 0,C 180,E1 28102.09,E2 28102.09} C_VEL
LIN {X 0,Y 578.814,Z 1121.865,A -85,B 0,C 180,E1 28100.952,E2 28100.952} C_VEL
LIN {X 0,Y 578.279,Z 1132.863,A -85,B 0,C 180,E1 28099.81,E2 28099.81} C_VEL
LIN {X 0,Y 577.749,Z 1143.271,A -85,B 0,C 180,E1 28098.464,E2 28098.464} C_VEL
LIN {X 0,Y 577.335,Z 1152.192,A -85,B 0,C 180,E1 28097.019,E2 28097.019} C_VEL
LIN {X 0,Y 577.02,Z 1159.464,A -85,B 0,C 180,E1 28095.478,E2 28095.478} C_VEL
LIN {X 0,Y 576.835,Z 1164.939,A -85,B 0,C 180,E1 28093.912,E2 28093.912} C_VEL
LIN {X 0,Y 576.739,Z 1168.62,A -85,B 0,C 180,E1 28092.313,E2 28092.313} C_VEL
LIN {X 0,Y 576.712,Z 1170.637,A -85,B 0,C 180,E1 28090.691,E2 28090.691} C_VEL
LIN {X 0,Y 576.757,Z 1170.891,A -85,B 0,C 180,E1 28089.077,E2 28089.077} C_VEL
LIN {X 0,Y 576.883,Z 1169.309,A -85,B 0,C 180,E1 28087.369,E2 28087.369} C_VEL
LIN {X 0,Y 577.078,Z 1166.026,A -85,B 0,C 180,E1 28085.768,E2 28085.768} C_VEL
LIN {X 0,Y 577.415,Z 1160.796,A -85,B 0,C 180,E1 28084.133,E2 28084.133} C_VEL
LIN {X 0,Y 577.844,Z 1154.334,A -85,B 0,C 180,E1 28082.678,E2 28082.678} C_VEL
LIN {X 0,Y 578.433,Z 1145.72,A -85,B 0,C 180,E1 28081.189,E2 28081.189} C_VEL
LIN {X 0,Y 579.092,Z 1136.322,A -85,B 0,C 180,E1 28079.901,E2 28079.901} C_VEL
LIN {X 0,Y 579.865,Z 1124.596,A -85,B 0,C 180,E1 28078.617,E2 28078.617} C_VEL
LIN {X 0,Y 580.631,Z 1112.271,A -85,B 0,C 180,E1 28077.533,E2 28077.533} C_VEL
LIN {X 0,Y 581.383,Z 1098.253,A -85,B 0,C 180,E1 28076.549,E2 28076.549} C_VEL
LIN {X 0,Y 582.064,Z 1083.924,A -85,B 0,C 180,E1 28075.764,E2 28075.764} C_VEL
LIN {X 0,Y 582.616,Z 1067.962,A -85,B 0,C 180,E1 28075.102,E2 28075.102} C_VEL
LIN {X 0,Y 582.958,Z 1051.951,A -85,B 0,C 180,E1 28074.636,E2 28074.636} C_VEL
LIN {X 0,Y 585.765,Z 973.919,A -85,B 0,C 180,E1 28073.07,E2 28073.07} C_VEL
LIN {X 0,Y 588.529,Z 912.884,A -85,B 0,C 180,E1 28071.869,E2 28071.869} C_VEL
LIN {X 0,Y 592.69,Z 865.839,A -85,B 0,C 180,E1 28068.024,E2 28068.024} C_VEL
LIN {X 0,Y 597.258,Z 824.173,A -85,B 0,C 180,E1 28064.513,E2 28064.513} C_VEL
LIN {X 0,Y 602.651,Z 784.674,A -85,B 0,C 180,E1 28061.073,E2 28061.073} C_VEL
LIN {X 0,Y 608.354,Z 750.634,A -85,B 0,C 180,E1 28057.992,E2 28057.992} C_VEL
LIN {X 0,Y 611.558,Z 732.104,A -85,B 0,C 180,E1 28056.181,E2 28056.181} C_VEL
LIN {X 0,Y 608.329,Z 721.821,A -85,B 0,C 180,E1 28054.249,E2 28054.249} C_VEL
LIN {X 0,Y 605.671,Z 713.845,A -85,B 0,C 180,E1 28052.435,E2 28052.435} C_VEL
LIN {X 0,Y 603.313,Z 707.221,A -85,B 0,C 180,E1 28050.466,E2 28050.466} C_VEL
LIN {X 0,Y 601.783,Z 703.271,A -85,B 0,C 180,E1 28048.775,E2 28048.775} C_VEL
LIN {X 0,Y 600.937,Z 700.385,A -85,B 0,C 180,E1 28046.582,E2 28046.582} C_VEL
LIN {X 0,Y 601.006,Z 699.88,A -85,B 0,C 180,E1 28045.552,E2 28045.552} C_VEL
LIN {X 0,Y 601.293,Z 700.349,A -85,B 0,C 180,E1 28044.402,E2 28044.402} C_VEL
LIN {X 0,Y 602.523,Z 703.616,A -85,B 0,C 180,E1 28042.33,E2 28042.33} C_VEL
LIN {X 0,Y 603.271,Z 705.057,A -85,B 0,C 180,E1 28041.692,E2 28041.692} C_VEL
LIN {X 0,Y 605.027,Z 709.164,A -85,B 0,C 180,E1 28040.362,E2 28040.362} C_VEL
LIN {X 0,Y 607.392,Z 714.998,A -85,B 0,C 180,E1 28038.941,E2 28038.941} C_VEL
LIN {X 0,Y 610.499,Z 723.987,A -85,B 0,C 180,E1 28037.307,E2 28037.307} C_VEL
LIN {X 0,Y 610.499,Z 725.121,A -85,B 0,C 180,E1 28037.18,E2 28037.18} C_VEL
LIN {X 0,Y 603.733,Z 759.473,A -85,B 0,C 180,E1 28034.669,E2 28034.669} C_VEL
LIN {X 0,Y 599.048,Z 793.61,A -85,B 0,C 180,E1 28032.27,E2 28032.27} C_VEL
LIN {X 0,Y 598.318,Z 814.461,A -85,B 0,C 180,E1 28030.735,E2 28030.735} C_VEL
LIN {X 0,Y 599.547,Z 831.941,A -85,B 0,C 180,E1 28029.376,E2 28029.376} C_VEL
LIN {X 0,Y 602.83,Z 848.481,A -85,B 0,C 180,E1 28028.013,E2 28028.013} C_VEL
LIN {X 0,Y 607.819,Z 862.874,A -85,B 0,C 180,E1 28026.761,E2 28026.761} C_VEL
LIN {X 0,Y 614.539,Z 876.098,A -85,B 0,C 180,E1 28025.557,E2 28025.557} C_VEL
LIN {X 0,Y 623.61,Z 888.922,A -85,B 0,C 180,E1 28024.335,E2 28024.335} C_VEL
LIN {X 0,Y 633.783,Z 899.685,A -85,B 0,C 180,E1 28023.263,E2 28023.263} C_VEL
LIN {X 0,Y 641.852,Z 906.9,A -85,B 0,C 180,E1 28022.532,E2 28022.532} C_VEL
LIN {X 0,Y 626.456,Z 930.191,A -85,B 0,C 180,E1 28021.889,E2 28021.889} C_VEL
LIN {X 0,Y 615.571,Z 949.483,A -85,B 0,C 180,E1 28021.261,E2 28021.261} C_VEL
LIN {X 0,Y 608.063,Z 965.836,A -85,B 0,C 180,E1 28020.646,E2 28020.646} C_VEL
LIN {X 0,Y 598.588,Z 987.46,A -85,B 0,C 180,E1 28019.796,E2 28019.796} C_VEL
LIN {X 0,Y 593.24,Z 1003.48,A -85,B 0,C 180,E1 28019.116,E2 28019.116} C_VEL
LIN {X 0,Y 591.106,Z 1025.004,A -85,B 0,C 180,E1 28018.903,E2 28018.903} C_VEL
LIN {X 0,Y 590.234,Z 1063.563,A -85,B 0,C 180,E1 28018.345,E2 28018.345} C_VEL
LIN {X 0,Y 589.351,Z 1085.407,A -85,B 0,C 180,E1 28017.86,E2 28017.86} C_VEL
LIN {X 0,Y 588.237,Z 1106.86,A -85,B 0,C 180,E1 28017.208,E2 28017.208} C_VEL
LIN {X 0,Y 586.904,Z 1128.968,A -85,B 0,C 180,E1 28016.345,E2 28016.345} C_VEL
LIN {X 0,Y 585.548,Z 1149.085,A -85,B 0,C 180,E1 28015.377,E2 28015.377} C_VEL
LIN {X 0,Y 584.151,Z 1168.365,A -85,B 0,C 180,E1 28014.254,E2 28014.254} C_VEL
LIN {X 0,Y 582.693,Z 1186.868,A -85,B 0,C 180,E1 28012.977,E2 28012.977} C_VEL
LIN {X 0,Y 581.336,Z 1204.609,A -85,B 0,C 180,E1 28011.542,E2 28011.542} C_VEL
LIN {X 0,Y 580.034,Z 1221.415,A -85,B 0,C 180,E1 28009.956,E2 28009.956} C_VEL
LIN {X 0,Y 578.869,Z 1237.016,A -85,B 0,C 180,E1 28008.217,E2 28008.217} C_VEL
LIN {X 0,Y 577.979,Z 1250.353,A -85,B 0,C 180,E1 28006.48,E2 28006.48} C_VEL
LIN {X 0,Y 577.25,Z 1262.445,A -85,B 0,C 180,E1 28004.647,E2 28004.647} C_VEL
LIN {X 0,Y 576.737,Z 1273.124,A -85,B 0,C 180,E1 28002.718,E2 28002.718} C_VEL
LIN {X 0,Y 576.357,Z 1282.38,A -85,B 0,C 180,E1 28000.696,E2 28000.696} C_VEL
LIN {X 0,Y 576.177,Z 1289.873,A -85,B 0,C 180,E1 27998.682,E2 27998.682} C_VEL
LIN {X 0,Y 576.082,Z 1295.628,A -85,B 0,C 180,E1 27996.677,E2 27996.677} C_VEL
LIN {X 0,Y 576.068,Z 1299.969,A -85,B 0,C 180,E1 27994.578,E2 27994.578} C_VEL
LIN {X 0,Y 576.074,Z 1302.72,A -85,B 0,C 180,E1 27992.486,E2 27992.486} C_VEL
LIN {X 0,Y 576.084,Z 1303.725,A -85,B 0,C 180,E1 27990.496,E2 27990.496} C_VEL
LIN {X 0,Y 576.094,Z 1303.2,A -85,B 0,C 180,E1 27988.308,E2 27988.308} C_VEL
LIN {X 0,Y 576.077,Z 1301.296,A -85,B 0,C 180,E1 27986.4,E2 27986.4} C_VEL
LIN {X 0,Y 576.074,Z 1297.705,A -85,B 0,C 180,E1 27984.321,E2 27984.321} C_VEL
LIN {X 0,Y 576.132,Z 1292.532,A -85,B 0,C 180,E1 27982.303,E2 27982.303} C_VEL
LIN {X 0,Y 576.279,Z 1285.069,A -85,B 0,C 180,E1 27980.108,E2 27980.108} C_VEL
LIN {X 0,Y 576.537,Z 1276.901,A -85,B 0,C 180,E1 27978.19,E2 27978.19} C_VEL
LIN {X 0,Y 576.972,Z 1266.283,A -85,B 0,C 180,E1 27976.162,E2 27976.162} C_VEL
LIN {X 0,Y 577.615,Z 1254.175,A -85,B 0,C 180,E1 27974.229,E2 27974.229} C_VEL
LIN {X 0,Y 578.525,Z 1239.324,A -85,B 0,C 180,E1 27972.236,E2 27972.236} C_VEL
LIN {X 0,Y 579.517,Z 1224.39,A -85,B 0,C 180,E1 27970.548,E2 27970.548} C_VEL
LIN {X 0,Y 580.694,Z 1208.074,A -85,B 0,C 180,E1 27968.95,E2 27968.95} C_VEL
LIN {X 0,Y 582.052,Z 1189.642,A -85,B 0,C 180,E1 27967.421,E2 27967.421} C_VEL
LIN {X 0,Y 583.432,Z 1171.132,A -85,B 0,C 180,E1 27966.102,E2 27966.102} C_VEL
LIN {X 0,Y 584.76,Z 1152.08,A -85,B 0,C 180,E1 27964.962,E2 27964.962} C_VEL
LIN {X 0,Y 586.21,Z 1130.762,A -85,B 0,C 180,E1 27963.891,E2 27963.891} C_VEL
LIN {X 0,Y 587.528,Z 1109.789,A -85,B 0,C 180,E1 27963.028,E2 27963.028} C_VEL
LIN {X 0,Y 588.688,Z 1087.748,A -85,B 0,C 180,E1 27962.322,E2 27962.322} C_VEL
LIN {X 0,Y 589.73,Z 1064.586,A -85,B 0,C 180,E1 27961.77,E2 27961.77} C_VEL
LIN {X 0,Y 590.395,Z 1040.85,A -85,B 0,C 180,E1 27961.384,E2 27961.384} C_VEL
LIN {X 0,Y 591.112,Z 1018.407,A -85,B 0,C 180,E1 27961.103,E2 27961.103} C_VEL
LIN {X 0,Y 591.315,Z 1016.296,A -85,B 0,C 180,E1 27961.077,E2 27961.077} C_VEL
LIN {X 0,Y 597.362,Z 997.022,A -85,B 0,C 180,E1 27960.189,E2 27960.189} C_VEL
LIN {X 0,Y 603.764,Z 980.642,A -85,B 0,C 180,E1 27959.495,E2 27959.495} C_VEL
LIN {X 0,Y 610.024,Z 967.013,A -85,B 0,C 180,E1 27958.968,E2 27958.968} C_VEL
LIN {X 0,Y 618.037,Z 950.073,A -85,B 0,C 180,E1 27958.337,E2 27958.337} C_VEL
LIN {X 0,Y 629.167,Z 930.743,A -85,B 0,C 180,E1 27957.723,E2 27957.723} C_VEL
LIN {X 0,Y 643.583,Z 908.785,A -85,B 0,C 180,E1 27957.137,E2 27957.137} C_VEL
LIN {X 0,Y 631.952,Z 898.409,A -85,B 0,C 180,E1 27956.005,E2 27956.005} C_VEL
LIN {X 0,Y 622.926,Z 887.853,A -85,B 0,C 180,E1 27954.948,E2 27954.948} C_VEL
LIN {X 0,Y 614.515,Z 874.755,A -85,B 0,C 180,E1 27953.731,E2 27953.731} C_VEL
LIN {X 0,Y 608.108,Z 860.765,A -85,B 0,C 180,E1 27952.527,E2 27952.527} C_VEL
LIN {X 0,Y 603.404,Z 845.557,A -85,B 0,C 180,E1 27951.306,E2 27951.306} C_VEL
LIN {X 0,Y 600.237,Z 827.834,A -85,B 0,C 180,E1 27949.983,E2 27949.983} C_VEL
LIN {X 0,Y 598.97,Z 807.153,A -85,B 0,C 180,E1 27948.551,E2 27948.551} C_VEL
LIN {X 0,Y 599.74,Z 783.195,A -85,B 0,C 180,E1 27947.008,E2 27947.008} C_VEL
LIN {X 0,Y 603.51,Z 735.599,A -85,B 0,C 180,E1 27944.023,E2 27944.023} C_VEL
LIN {X 0,Y 604.518,Z 721.109,A -85,B 0,C 180,E1 27943.088,E2 27943.088} C_VEL
LIN {X 0,Y 593.262,Z 695.594,A -85,B 0,C 180,E1 27940.331,E2 27940.331} C_VEL
LIN {X 0,Y 585.519,Z 678.842,A -85,B 0,C 180,E1 27938.386,E2 27938.386} C_VEL
LIN {X 0,Y 586.802,Z 679.117,A -85,B 0,C 180,E1 27938.151,E2 27938.151} C_VEL
LIN {X 0,Y 591.006,Z 689.856,A -85,B 0,C 180,E1 27936.43,E2 27936.43} C_VEL
LIN {X 0,Y 594.531,Z 701.629,A -85,B 0,C 180,E1 27934.842,E2 27934.842} C_VEL
LIN {X 0,Y 596.109,Z 708.993,A -85,B 0,C 180,E1 27933.957,E2 27933.957} C_VEL
LIN {X 0,Y 596.124,Z 711.842,A -85,B 0,C 180,E1 27933.738,E2 27933.738} C_VEL
LIN {X 0,Y 599.931,Z 730.463,A -85,B 0,C 180,E1 27932.938,E2 27932.938} C_VEL
LIN {X 0,Y 600.574,Z 735.656,A -85,B 0,C 180,E1 27932.761,E2 27932.761} C_VEL
LIN {X 0,Y 595.619,Z 840.058,A -85,B 0,C 180,E1 27930.96,E2 27930.96} C_VEL
LIN {X 0,Y 592.393,Z 938.256,A -85,B 0,C 180,E1 27929.401,E2 27929.401} C_VEL
LIN {X 0,Y 590.579,Z 1012.951,A -85,B 0,C 180,E1 27928.278,E2 27928.278} C_VEL
LIN {X 0,Y 589.77,Z 1035.334,A -85,B 0,C 180,E1 27927.762,E2 27927.762} C_VEL
LIN {X 0,Y 588.754,Z 1057.431,A -85,B 0,C 180,E1 27927.075,E2 27927.075} C_VEL
LIN {X 0,Y 587.609,Z 1078.074,A -85,B 0,C 180,E1 27926.259,E2 27926.259} C_VEL
LIN {X 0,Y 586.278,Z 1099.024,A -85,B 0,C 180,E1 27925.238,E2 27925.238} C_VEL
LIN {X 0,Y 584.866,Z 1118.432,A -85,B 0,C 180,E1 27924.086,E2 27924.086} C_VEL
LIN {X 0,Y 583.429,Z 1137.042,A -85,B 0,C 180,E1 27922.774,E2 27922.774} C_VEL
LIN {X 0,Y 581.997,Z 1154.728,A -85,B 0,C 180,E1 27921.307,E2 27921.307} C_VEL
LIN {X 0,Y 580.667,Z 1170.979,A -85,B 0,C 180,E1 27919.725,E2 27919.725} C_VEL
LIN {X 0,Y 579.488,Z 1185.505,A -85,B 0,C 180,E1 27918.058,E2 27918.058} C_VEL
LIN {X 0,Y 578.445,Z 1198.858,A -85,B 0,C 180,E1 27916.262,E2 27916.262} C_VEL
LIN {X 0,Y 577.585,Z 1210.972,A -85,B 0,C 180,E1 27914.333,E2 27914.333} C_VEL
LIN {X 0,Y 576.956,Z 1221.128,A -85,B 0,C 180,E1 27912.41,E2 27912.41} C_VEL
LIN {X 0,Y 576.51,Z 1229.771,A -85,B 0,C 180,E1 27910.392,E2 27910.392} C_VEL
LIN {X 0,Y 576.215,Z 1237.001,A -85,B 0,C 180,E1 27908.281,E2 27908.281} C_VEL
LIN {X 0,Y 576.059,Z 1242.502,A -85,B 0,C 180,E1 27906.178,E2 27906.178} C_VEL
LIN {X 0,Y 575.976,Z 1246.28,A -85,B 0,C 180,E1 27904.082,E2 27904.082} C_VEL
LIN {X 0,Y 575.95,Z 1248.549,A -85,B 0,C 180,E1 27901.89,E2 27901.89} C_VEL
LIN {X 0,Y 575.955,Z 1249.206,A -85,B 0,C 180,E1 27899.801,E2 27899.801} C_VEL
LIN {X 0,Y 575.948,Z 1248.269,A -85,B 0,C 180,E1 27897.712,E2 27897.712} C_VEL
LIN {X 0,Y 575.977,Z 1245.648,A -85,B 0,C 180,E1 27895.519,E2 27895.519} C_VEL
LIN {X 0,Y 576.063,Z 1241.583,A -85,B 0,C 180,E1 27893.422,E2 27893.422} C_VEL
LIN {X 0,Y 576.218,Z 1235.796,A -85,B 0,C 180,E1 27891.317,E2 27891.317} C_VEL
LIN {X 0,Y 576.529,Z 1228.215,A -85,B 0,C 180,E1 27889.204,E2 27889.204} C_VEL
LIN {X 0,Y 577.044,Z 1218.711,A -85,B 0,C 180,E1 27887.084,E2 27887.084} C_VEL
LIN {X 0,Y 577.727,Z 1208.286,A -85,B 0,C 180,E1 27885.158,E2 27885.158} C_VEL
LIN {X 0,Y 578.586,Z 1196.408,A -85,B 0,C 180,E1 27883.329,E2 27883.329} C_VEL
LIN {X 0,Y 579.696,Z 1182.439,A -85,B 0,C 180,E1 27881.496,E2 27881.496} C_VEL
LIN {X 0,Y 580.962,Z 1167.634,A -85,B 0,C 180,E1 27879.833,E2 27879.833} C_VEL
LIN {X 0,Y 582.362,Z 1151.248,A -85,B 0,C 180,E1 27878.261,E2 27878.261} C_VEL
LIN {X 0,Y 583.819,Z 1134.016,A -85,B 0,C 180,E1 27876.855,E2 27876.855} C_VEL
LIN {X 0,Y 585.377,Z 1114.966,A -85,B 0,C 180,E1 27875.53,E2 27875.53} C_VEL
LIN {X 0,Y 586.833,Z 1095.893,A -85,B 0,C 180,E1 27874.41,E2 27874.41} C_VEL
LIN {X 0,Y 588.256,Z 1075.282,A -85,B 0,C 180,E1 27873.412,E2 27873.412} C_VEL
LIN {X 0,Y 589.479,Z 1054.722,A -85,B 0,C 180,E1 27872.606,E2 27872.606} C_VEL
LIN {X 0,Y 590.563,Z 1032.352,A -85,B 0,C 180,E1 27871.917,E2 27871.917} C_VEL
LIN {X 0,Y 591.453,Z 1010.155,A -85,B 0,C 180,E1 27871.417,E2 27871.417} C_VEL
LIN {X 0,Y 592.282,Z 971.651,A -85,B 0,C 180,E1 27870.857,E2 27870.857} C_VEL
LIN {X 0,Y 596.996,Z 757.754,A -85,B 0,C 180,E1 27867.883,E2 27867.883} C_VEL
LIN {X 0,Y 597.403,Z 732.969,A -85,B 0,C 180,E1 27867.519,E2 27867.519} C_VEL
LIN {X 0,Y 590.882,Z 703.21,A -85,B 0,C 180,E1 27866.635,E2 27866.635} C_VEL
LIN {X 0,Y 587.815,Z 692.137,A -85,B 0,C 180,E1 27865.417,E2 27865.417} C_VEL
LIN {X 0,Y 580.181,Z 669.226,A -85,B 0,C 180,E1 27862.771,E2 27862.771} C_VEL
LIN {X 0,Y 577.309,Z 660.756,A -85,B 0,C 180,E1 27861.743,E2 27861.743} C_VEL
LIN {X 0,Y 577.316,Z 660.757,A -85,B 0,C 180,E1 27861.121,E2 27861.121} C_VEL
LIN {X 0,Y 576.366,Z 660.873,A -85,B 0,C 180,E1 27860.356,E2 27860.356} C_VEL
LIN {X 0,Y 569.83,Z 661.69,A -85,B 0,C 180,E1 27858.155,E2 27858.155} C_VEL
LIN {X 0,Y 569.373,Z 661.745,A -85,B 0,C 180,E1 27857.652,E2 27857.652} C_VEL
LIN {X 0,Y 569.367,Z 661.746,A -85,B 0,C 180,E1 27854.343,E2 27854.343} C_VEL
LIN {X 0,Y 569.366,Z 661.748,A -85,B 0,C 180,E1 27851.057,E2 27851.057} C_VEL
LIN {X 0,Y 569.384,Z 661.742,A -85,B 0,C 180,E1 27847.791,E2 27847.791} C_VEL
LIN {X 0,Y 569.375,Z 661.742,A -85,B 0,C 180,E1 27844.436,E2 27844.436} C_VEL
LIN {X 0,Y 569.388,Z 661.74,A -85,B 0,C 180,E1 27841.085,E2 27841.085} C_VEL
LIN {X 0,Y 569.367,Z 661.742,A -85,B 0,C 180,E1 27837.736,E2 27837.736} C_VEL
LIN {X 0,Y 569.366,Z 661.743,A -85,B 0,C 180,E1 27834.486,E2 27834.486} C_VEL
LIN {X 0,Y 569.369,Z 661.743,A -85,B 0,C 180,E1 27831.21,E2 27831.21} C_VEL
LIN {X 0,Y 569.376,Z 661.743,A -85,B 0,C 180,E1 27827.858,E2 27827.858} C_VEL
LIN {X 0,Y 569.376,Z 661.741,A -85,B 0,C 180,E1 27824.441,E2 27824.441} C_VEL
LIN {X 0,Y 569.381,Z 661.746,A -85,B 0,C 180,E1 27821.139,E2 27821.139} C_VEL
LIN {X 0,Y 569.383,Z 661.736,A -85,B 0,C 180,E1 27817.773,E2 27817.773} C_VEL
LIN {X 0,Y 569.365,Z 661.742,A -85,B 0,C 180,E1 27814.534,E2 27814.534} C_VEL
LIN {X 0,Y 569.374,Z 661.742,A -85,B 0,C 180,E1 27811.209,E2 27811.209} C_VEL
LIN {X 0,Y 569.374,Z 661.742,A -85,B 0,C 180,E1 27807.764,E2 27807.764} C_VEL
LIN {X 0,Y 569.368,Z 661.743,A -85,B 0,C 180,E1 27804.459,E2 27804.459} C_VEL
LIN {X 0,Y 569.364,Z 661.746,A -85,B 0,C 180,E1 27801.213,E2 27801.213} C_VEL
LIN {X 0,Y 569.382,Z 661.744,A -85,B 0,C 180,E1 27797.939,E2 27797.939} C_VEL
LIN {X 0,Y 569.376,Z 661.745,A -85,B 0,C 180,E1 27794.604,E2 27794.604} C_VEL
LIN {X 0,Y 569.383,Z 661.745,A -85,B 0,C 180,E1 27791.256,E2 27791.256} C_VEL
LIN {X 0,Y 569.374,Z 661.744,A -85,B 0,C 180,E1 27787.927,E2 27787.927} C_VEL
LIN {X 0,Y 569.367,Z 661.741,A -85,B 0,C 180,E1 27784.63,E2 27784.63} C_VEL
LIN {X 0,Y 569.366,Z 661.744,A -85,B 0,C 180,E1 27781.354,E2 27781.354} C_VEL
LIN {X 0,Y 569.369,Z 661.733,A -85,B 0,C 180,E1 27778.091,E2 27778.091} C_VEL
LIN {X 0,Y 569.381,Z 661.736,A -85,B 0,C 180,E1 27774.709,E2 27774.709} C_VEL
LIN {X 0,Y 569.387,Z 661.736,A -85,B 0,C 180,E1 27771.308,E2 27771.308} C_VEL
LIN {X 0,Y 569.382,Z 661.735,A -85,B 0,C 180,E1 27767.946,E2 27767.946} C_VEL
LIN {X 0,Y 569.39,Z 661.798,A -85,B 0,C 180,E1 27767.872,E2 27767.872} C_VEL
LIN {X 0,Y 578.926,Z 687.513,A -85,B 0,C 180,E1 27764.85,E2 27764.85} C_VEL
LIN {X 0,Y 586.656,Z 709.824,A -85,B 0,C 180,E1 27762.406,E2 27762.406} C_VEL
LIN {X 0,Y 584.386,Z 745.122,A -85,B 0,C 180,E1 27759.595,E2 27759.595} C_VEL
LIN {X 0,Y 581.682,Z 787.114,A -85,B 0,C 180,E1 27756.306,E2 27756.306} C_VEL
LIN {X 0,Y 579.174,Z 830.342,A -85,B 0,C 180,E1 27752.966,E2 27752.966} C_VEL
LIN {X 0,Y 576.806,Z 876.695,A -85,B 0,C 180,E1 27749.436,E2 27749.436} C_VEL
LIN {X 0,Y 575.701,Z 902.975,A -85,B 0,C 180,E1 27747.487,E2 27747.487} C_VEL
LIN {X 0,Y 576.573,Z 912.018,A -85,B 0,C 180,E1 27747.305,E2 27747.305} C_VEL
LIN {X 0,Y 573.658,Z 1047.58,A -85,B 0,C 180,E1 27745.08,E2 27745.08} C_VEL
LIN {X 0,Y 573.328,Z 1064.577,A -85,B 0,C 180,E1 27744.607,E2 27744.607} C_VEL
LIN {X 0,Y 572.867,Z 1079.927,A -85,B 0,C 180,E1 27743.997,E2 27743.997} C_VEL
LIN {X 0,Y 572.238,Z 1095.806,A -85,B 0,C 180,E1 27743.151,E2 27743.151} C_VEL
LIN {X 0,Y 571.617,Z 1109.713,A -85,B 0,C 180,E1 27742.2,E2 27742.2} C_VEL
LIN {X 0,Y 570.943,Z 1123.329,A -85,B 0,C 180,E1 27741.029,E2 27741.029} C_VEL
LIN {X 0,Y 570.344,Z 1134.966,A -85,B 0,C 180,E1 27739.777,E2 27739.777} C_VEL
LIN {X 0,Y 569.809,Z 1145.17,A -85,B 0,C 180,E1 27738.413,E2 27738.413} C_VEL
LIN {X 0,Y 569.38,Z 1153.842,A -85,B 0,C 180,E1 27736.949,E2 27736.949} C_VEL
LIN {X 0,Y 569.068,Z 1160.969,A -85,B 0,C 180,E1 27735.386,E2 27735.386} C_VEL
LIN {X 0,Y 568.886,Z 1166.175,A -85,B 0,C 180,E1 27733.83,E2 27733.83} C_VEL
LIN {X 0,Y 568.786,Z 1169.994,A -85,B 0,C 180,E1 27732.075,E2 27732.075} C_VEL
LIN {X 0,Y 568.773,Z 1171.747,A -85,B 0,C 180,E1 27730.432,E2 27730.432} C_VEL
LIN {X 0,Y 568.846,Z 1171.714,A -85,B 0,C 180,E1 27728.695,E2 27728.695} C_VEL
LIN {X 0,Y 568.98,Z 1169.927,A -85,B 0,C 180,E1 27727.066,E2 27727.066} C_VEL
LIN {X 0,Y 569.242,Z 1166.131,A -85,B 0,C 180,E1 27725.342,E2 27725.342} C_VEL
LIN {X 0,Y 569.627,Z 1160.648,A -85,B 0,C 180,E1 27723.724,E2 27723.724} C_VEL
LIN {X 0,Y 570.171,Z 1153.169,A -85,B 0,C 180,E1 27722.111,E2 27722.111} C_VEL
LIN {X 0,Y 570.809,Z 1144.607,A -85,B 0,C 180,E1 27720.703,E2 27720.703} C_VEL
LIN {X 0,Y 571.621,Z 1133.89,A -85,B 0,C 180,E1 27719.298,E2 27719.298} C_VEL
LIN {X 0,Y 572.457,Z 1121.799,A -85,B 0,C 180,E1 27718.048,E2 27718.048} C_VEL
LIN {X 0,Y 573.251,Z 1109.288,A -85,B 0,C 180,E1 27717,E2 27717} C_VEL
LIN {X 0,Y 574.039,Z 1095.003,A -85,B 0,C 180,E1 27716.055,E2 27716.055} C_VEL
LIN {X 0,Y 574.729,Z 1080.714,A -85,B 0,C 180,E1 27715.31,E2 27715.31} C_VEL
LIN {X 0,Y 575.256,Z 1064.642,A -85,B 0,C 180,E1 27714.689,E2 27714.689} C_VEL
LIN {X 0,Y 575.594,Z 1048.468,A -85,B 0,C 180,E1 27714.255,E2 27714.255} C_VEL
LIN {X 0,Y 581.558,Z 914.231,A -85,B 0,C 180,E1 27711.497,E2 27711.497} C_VEL
LIN {X 0,Y 585.946,Z 867.59,A -85,B 0,C 180,E1 27707.634,E2 27707.634} C_VEL
LIN {X 0,Y 590.97,Z 825.007,A -85,B 0,C 180,E1 27703.991,E2 27703.991} C_VEL
LIN {X 0,Y 596.893,Z 784.753,A -85,B 0,C 180,E1 27700.425,E2 27700.425} C_VEL
LIN {X 0,Y 602.612,Z 753.23,A -85,B 0,C 180,E1 27697.514,E2 27697.514} C_VEL
LIN {X 0,Y 605.731,Z 736.815,A -85,B 0,C 180,E1 27695.896,E2 27695.896} C_VEL
LIN {X 0,Y 602.701,Z 726.68,A -85,B 0,C 180,E1 27693.919,E2 27693.919} C_VEL
LIN {X 0,Y 600.235,Z 719.104,A -85,B 0,C 180,E1 27692.089,E2 27692.089} C_VEL
LIN {X 0,Y 598.373,Z 713.398,A -85,B 0,C 180,E1 27690.33,E2 27690.33} C_VEL
LIN {X 0,Y 597.095,Z 709.734,A -85,B 0,C 180,E1 27688.726,E2 27688.726} C_VEL
LIN {X 0,Y 596.374,Z 706.798,A -85,B 0,C 180,E1 27686.407,E2 27686.407} C_VEL
LIN {X 0,Y 596.61,Z 706.559,A -85,B 0,C 180,E1 27685.028,E2 27685.028} C_VEL
LIN {X 0,Y 596.819,Z 707.55,A -85,B 0,C 180,E1 27683.981,E2 27683.981} C_VEL
LIN {X 0,Y 598.447,Z 710.835,A -85,B 0,C 180,E1 27681.997,E2 27681.997} C_VEL
LIN {X 0,Y 600.355,Z 715.87,A -85,B 0,C 180,E1 27680.365,E2 27680.365} C_VEL
LIN {X 0,Y 602.462,Z 721.325,A -85,B 0,C 180,E1 27679.036,E2 27679.036} C_VEL
LIN {X 0,Y 604.977,Z 729.066,A -85,B 0,C 180,E1 27677.597,E2 27677.597} C_VEL
LIN {X 0,Y 597.831,Z 762.387,A -85,B 0,C 180,E1 27675.105,E2 27675.105} C_VEL
LIN {X 0,Y 592.861,Z 795.171,A -85,B 0,C 180,E1 27672.75,E2 27672.75} C_VEL
LIN {X 0,Y 591.765,Z 816.364,A -85,B 0,C 180,E1 27671.155,E2 27671.155} C_VEL
LIN {X 0,Y 592.76,Z 834.458,A -85,B 0,C 180,E1 27669.718,E2 27669.718} C_VEL
LIN {X 0,Y 595.971,Z 851.738,A -85,B 0,C 180,E1 27668.262,E2 27668.262} C_VEL
LIN {X 0,Y 601.165,Z 867.07,A -85,B 0,C 180,E1 27666.899,E2 27666.899} C_VEL
LIN {X 0,Y 607.9,Z 880.458,A -85,B 0,C 180,E1 27665.654,E2 27665.654} C_VEL
LIN {X 0,Y 616.877,Z 893.316,A -85,B 0,C 180,E1 27664.408,E2 27664.408} C_VEL
LIN {X 0,Y 627.65,Z 904.85,A -85,B 0,C 180,E1 27663.242,E2 27663.242} C_VEL
LIN {X 0,Y 632.245,Z 909.281,A -85,B 0,C 180,E1 27662.8,E2 27662.8} C_VEL
LIN {X 0,Y 617.746,Z 931.741,A -85,B 0,C 180,E1 27662.163,E2 27662.163} C_VEL
LIN {X 0,Y 607.65,Z 950.13,A -85,B 0,C 180,E1 27661.55,E2 27661.55} C_VEL
LIN {X 0,Y 591.805,Z 985.637,A -85,B 0,C 180,E1 27660.173,E2 27660.173} C_VEL
LIN {X 0,Y 586.206,Z 1002.169,A -85,B 0,C 180,E1 27659.467,E2 27659.467} C_VEL
LIN {X 0,Y 583.944,Z 1023.962,A -85,B 0,C 180,E1 27659.253,E2 27659.253} C_VEL
LIN {X 0,Y 582.961,Z 1063.287,A -85,B 0,C 180,E1 27658.676,E2 27658.676} C_VEL
LIN {X 0,Y 582.035,Z 1085.052,A -85,B 0,C 180,E1 27658.186,E2 27658.186} C_VEL
LIN {X 0,Y 580.866,Z 1106.501,A -85,B 0,C 180,E1 27657.526,E2 27657.526} C_VEL
LIN {X 0,Y 579.464,Z 1128.606,A -85,B 0,C 180,E1 27656.655,E2 27656.655} C_VEL
LIN {X 0,Y 578.056,Z 1148.579,A -85,B 0,C 180,E1 27655.683,E2 27655.683} C_VEL
LIN {X 0,Y 576.511,Z 1168.823,A -85,B 0,C 180,E1 27654.487,E2 27654.487} C_VEL
LIN {X 0,Y 574.99,Z 1187.229,A -85,B 0,C 180,E1 27653.194,E2 27653.194} C_VEL
LIN {X 0,Y 573.512,Z 1205.579,A -85,B 0,C 180,E1 27651.679,E2 27651.679} C_VEL
LIN {X 0,Y 572.208,Z 1221.633,A -85,B 0,C 180,E1 27650.134,E2 27650.134} C_VEL
LIN {X 0,Y 571.049,Z 1236.318,A -85,B 0,C 180,E1 27648.475,E2 27648.475} C_VEL
LIN {X 0,Y 570.057,Z 1250.459,A -85,B 0,C 180,E1 27646.611,E2 27646.611} C_VEL
LIN {X 0,Y 569.258,Z 1263.084,A -85,B 0,C 180,E1 27644.649,E2 27644.649} C_VEL
LIN {X 0,Y 568.72,Z 1273.962,A -85,B 0,C 180,E1 27642.638,E2 27642.638} C_VEL
LIN {X 0,Y 568.35,Z 1282.755,A -85,B 0,C 180,E1 27640.644,E2 27640.644} C_VEL
LIN {X 0,Y 568.168,Z 1290.415,A -85,B 0,C 180,E1 27638.49,E2 27638.49} C_VEL
LIN {X 0,Y 568.082,Z 1296.003,A -85,B 0,C 180,E1 27636.466,E2 27636.466} C_VEL
LIN {X 0,Y 568.08,Z 1300.077,A -85,B 0,C 180,E1 27634.339,E2 27634.339} C_VEL
LIN {X 0,Y 568.085,Z 1302.621,A -85,B 0,C 180,E1 27632.117,E2 27632.117} C_VEL
LIN {X 0,Y 568.111,Z 1303.448,A -85,B 0,C 180,E1 27629.999,E2 27629.999} C_VEL
LIN {X 0,Y 568.093,Z 1302.521,A -85,B 0,C 180,E1 27627.88,E2 27627.88} C_VEL
LIN {X 0,Y 568.085,Z 1300.054,A -85,B 0,C 180,E1 27625.759,E2 27625.759} C_VEL
LIN {X 0,Y 568.096,Z 1295.904,A -85,B 0,C 180,E1 27623.632,E2 27623.632} C_VEL
LIN {X 0,Y 568.17,Z 1290.22,A -85,B 0,C 180,E1 27621.6,E2 27621.6} C_VEL
LIN {X 0,Y 568.335,Z 1282.508,A -85,B 0,C 180,E1 27619.456,E2 27619.456} C_VEL
LIN {X 0,Y 568.691,Z 1273.071,A -85,B 0,C 180,E1 27617.376,E2 27617.376} C_VEL
LIN {X 0,Y 569.212,Z 1261.803,A -85,B 0,C 180,E1 27615.346,E2 27615.346} C_VEL
LIN {X 0,Y 569.958,Z 1248.74,A -85,B 0,C 180,E1 27613.383,E2 27613.383} C_VEL
LIN {X 0,Y 570.847,Z 1235.033,A -85,B 0,C 180,E1 27611.621,E2 27611.621} C_VEL
LIN {X 0,Y 571.926,Z 1220.136,A -85,B 0,C 180,E1 27609.96,E2 27609.96} C_VEL
LIN {X 0,Y 573.22,Z 1203.154,A -85,B 0,C 180,E1 27608.349,E2 27608.349} C_VEL
LIN {X 0,Y 574.47,Z 1186.714,A -85,B 0,C 180,E1 27607.003,E2 27607.003} C_VEL
LIN {X 0,Y 575.978,Z 1167.446,A -85,B 0,C 180,E1 27605.65,E2 27605.65} C_VEL
LIN {X 0,Y 577.383,Z 1148.253,A -85,B 0,C 180,E1 27604.51,E2 27604.51} C_VEL
LIN {X 0,Y 578.839,Z 1127.338,A -85,B 0,C 180,E1 27603.483,E2 27603.483} C_VEL
LIN {X 0,Y 580.181,Z 1106.217,A -85,B 0,C 180,E1 27602.633,E2 27602.633} C_VEL
LIN {X 0,Y 581.448,Z 1083.476,A -85,B 0,C 180,E1 27601.919,E2 27601.919} C_VEL
LIN {X 0,Y 582.48,Z 1060.049,A -85,B 0,C 180,E1 27601.388,E2 27601.388} C_VEL
LIN {X 0,Y 583.213,Z 1028.705,A -85,B 0,C 180,E1 27600.918,E2 27600.918} C_VEL
LIN {X 0,Y 584.123,Z 1015.267,A -85,B 0,C 180,E1 27600.743,E2 27600.743} C_VEL
LIN {X 0,Y 590.836,Z 994.359,A -85,B 0,C 180,E1 27599.769,E2 27599.769} C_VEL
LIN {X 0,Y 597.432,Z 978.051,A -85,B 0,C 180,E1 27599.081,E2 27599.081} C_VEL
LIN {X 0,Y 603.36,Z 965.237,A -85,B 0,C 180,E1 27598.581,E2 27598.581} C_VEL
LIN {X 0,Y 611.421,Z 948.377,A -85,B 0,C 180,E1 27597.948,E2 27597.948} C_VEL
LIN {X 0,Y 622.997,Z 928.366,A -85,B 0,C 180,E1 27597.311,E2 27597.311} C_VEL
LIN {X 0,Y 634.164,Z 911.361,A -85,B 0,C 180,E1 27596.849,E2 27596.849} C_VEL
LIN {X 0,Y 623.199,Z 900.78,A -85,B 0,C 180,E1 27595.72,E2 27595.72} C_VEL
LIN {X 0,Y 613.791,Z 888.796,A -85,B 0,C 180,E1 27594.54,E2 27594.54} C_VEL
LIN {X 0,Y 605.962,Z 875.441,A -85,B 0,C 180,E1 27593.316,E2 27593.316} C_VEL
LIN {X 0,Y 599.6,Z 860.001,A -85,B 0,C 180,E1 27592.002,E2 27592.002} C_VEL
LIN {X 0,Y 595.221,Z 843.393,A -85,B 0,C 180,E1 27590.684,E2 27590.684} C_VEL
LIN {X 0,Y 592.714,Z 825.598,A -85,B 0,C 180,E1 27589.369,E2 27589.369} C_VEL
LIN {X 0,Y 591.992,Z 803.109,A -85,B 0,C 180,E1 27587.825,E2 27587.825} C_VEL
LIN {X 0,Y 594.251,Z 767.786,A -85,B 0,C 180,E1 27585.575,E2 27585.575} C_VEL
LIN {X 0,Y 597.856,Z 724.846,A -85,B 0,C 180,E1 27582.833,E2 27582.833} C_VEL
LIN {X 0,Y 586.761,Z 699.679,A -85,B 0,C 180,E1 27580.08,E2 27580.08} C_VEL
LIN {X 0,Y 580.505,Z 685.71,A -85,B 0,C 180,E1 27578.433,E2 27578.433} C_VEL
LIN {X 0,Y 582.019,Z 685.984,A -85,B 0,C 180,E1 27578.149,E2 27578.149} C_VEL
LIN {X 0,Y 585.749,Z 696.194,A -85,B 0,C 180,E1 27576.484,E2 27576.484} C_VEL
LIN {X 0,Y 588.891,Z 707.748,A -85,B 0,C 180,E1 27574.904,E2 27574.904} C_VEL
LIN {X 0,Y 590.073,Z 712.674,A -85,B 0,C 180,E1 27574.323,E2 27574.323} C_VEL
LIN {X 0,Y 593.863,Z 731.816,A -85,B 0,C 180,E1 27573.448,E2 27573.448} C_VEL
LIN {X 0,Y 594.554,Z 737.42,A -85,B 0,C 180,E1 27573.25,E2 27573.25} C_VEL
LIN {X 0,Y 589.296,Z 835.828,A -85,B 0,C 180,E1 27571.486,E2 27571.486} C_VEL
LIN {X 0,Y 585.675,Z 932.602,A -85,B 0,C 180,E1 27569.887,E2 27569.887} C_VEL
LIN {X 0,Y 583.43,Z 1014.32,A -85,B 0,C 180,E1 27568.614,E2 27568.614} C_VEL
LIN {X 0,Y 582.554,Z 1036.883,A -85,B 0,C 180,E1 27568.075,E2 27568.075} C_VEL
LIN {X 0,Y 581.481,Z 1058.462,A -85,B 0,C 180,E1 27567.386,E2 27567.386} C_VEL
LIN {X 0,Y 580.2,Z 1080.029,A -85,B 0,C 180,E1 27566.51,E2 27566.51} C_VEL
LIN {X 0,Y 578.875,Z 1099.758,A -85,B 0,C 180,E1 27565.529,E2 27565.529} C_VEL
LIN {X 0,Y 577.365,Z 1119.438,A -85,B 0,C 180,E1 27564.342,E2 27564.342} C_VEL
LIN {X 0,Y 575.882,Z 1137.613,A -85,B 0,C 180,E1 27563.04,E2 27563.04} C_VEL
LIN {X 0,Y 574.365,Z 1155.312,A -85,B 0,C 180,E1 27561.551,E2 27561.551} C_VEL
LIN {X 0,Y 573.016,Z 1171.08,A -85,B 0,C 180,E1 27560,E2 27560} C_VEL
LIN {X 0,Y 571.721,Z 1186.089,A -85,B 0,C 180,E1 27558.256,E2 27558.256} C_VEL
LIN {X 0,Y 570.648,Z 1199.046,A -85,B 0,C 180,E1 27556.491,E2 27556.491} C_VEL
LIN {X 0,Y 569.728,Z 1211.218,A -85,B 0,C 180,E1 27554.535,E2 27554.535} C_VEL
LIN {X 0,Y 569.053,Z 1221.397,A -85,B 0,C 180,E1 27552.585,E2 27552.585} C_VEL
LIN {X 0,Y 568.572,Z 1230.077,A -85,B 0,C 180,E1 27550.538,E2 27550.538} C_VEL
LIN {X 0,Y 568.248,Z 1237.346,A -85,B 0,C 180,E1 27548.398,E2 27548.398} C_VEL
LIN {X 0,Y 568.082,Z 1242.868,A -85,B 0,C 180,E1 27546.265,E2 27546.265} C_VEL
LIN {X 0,Y 567.99,Z 1246.655,A -85,B 0,C 180,E1 27544.139,E2 27544.139} C_VEL
LIN {X 0,Y 567.956,Z 1248.867,A -85,B 0,C 180,E1 27542.018,E2 27542.018} C_VEL
LIN {X 0,Y 567.967,Z 1249.608,A -85,B 0,C 180,E1 27539.899,E2 27539.899} C_VEL
LIN {X 0,Y 567.957,Z 1248.702,A -85,B 0,C 180,E1 27537.78,E2 27537.78} C_VEL
LIN {X 0,Y 567.987,Z 1246.15,A -85,B 0,C 180,E1 27535.558,E2 27535.558} C_VEL
LIN {X 0,Y 568.078,Z 1242.144,A -85,B 0,C 180,E1 27533.43,E2 27533.43} C_VEL
LIN {X 0,Y 568.242,Z 1236.372,A -85,B 0,C 180,E1 27531.296,E2 27531.296} C_VEL
LIN {X 0,Y 568.57,Z 1228.842,A -85,B 0,C 180,E1 27529.154,E2 27529.154} C_VEL
LIN {X 0,Y 569.077,Z 1219.901,A -85,B 0,C 180,E1 27527.106,E2 27527.106} C_VEL
LIN {X 0,Y 569.825,Z 1208.983,A -85,B 0,C 180,E1 27525.052,E2 27525.052} C_VEL
LIN {X 0,Y 570.724,Z 1197.14,A -85,B 0,C 180,E1 27523.197,E2 27523.197} C_VEL
LIN {X 0,Y 571.886,Z 1183.236,A -85,B 0,C 180,E1 27521.339,E2 27521.339} C_VEL
LIN {X 0,Y 573.185,Z 1168.822,A -85,B 0,C 180,E1 27519.687,E2 27519.687} C_VEL
LIN {X 0,Y 574.587,Z 1152.929,A -85,B 0,C 180,E1 27518.136,E2 27518.136} C_VEL
LIN {X 0,Y 576.125,Z 1135.629,A -85,B 0,C 180,E1 27516.69,E2 27516.69} C_VEL
LIN {X 0,Y 577.673,Z 1117.613,A -85,B 0,C 180,E1 27515.4,E2 27515.4} C_VEL
LIN {X 0,Y 579.252,Z 1097.99,A -85,B 0,C 180,E1 27514.215,E2 27514.215} C_VEL
LIN {X 0,Y 580.671,Z 1078.294,A -85,B 0,C 180,E1 27513.232,E2 27513.232} C_VEL
LIN {X 0,Y 582.032,Z 1057.071,A -85,B 0,C 180,E1 27512.365,E2 27512.365} C_VEL
LIN {X 0,Y 583.17,Z 1035.66,A -85,B 0,C 180,E1 27511.672,E2 27511.672} C_VEL
LIN {X 0,Y 584.09,Z 1013.444,A -85,B 0,C 180,E1 27511.145,E2 27511.145} C_VEL
LIN {X 0,Y 584.806,Z 986.042,A -85,B 0,C 180,E1 27510.712,E2 27510.712} C_VEL
LIN {X 0,Y 589.527,Z 780.195,A -85,B 0,C 180,E1 27507.809,E2 27507.809} C_VEL
LIN {X 0,Y 590.559,Z 734.637,A -85,B 0,C 180,E1 27507.142,E2 27507.142} C_VEL
LIN {X 0,Y 583.912,Z 705.329,A -85,B 0,C 180,E1 27506.263,E2 27506.263} C_VEL
LIN {X 0,Y 583.136,Z 703.535,A -85,B 0,C 180,E1 27506.169,E2 27506.169} C_VEL
LIN {X 0,Y 576.638,Z 683.018,A -85,B 0,C 180,E1 27503.822,E2 27503.822} C_VEL
LIN {X 0,Y 569.369,Z 661.748,A -85,B 0,C 180,E1 27501.272,E2 27501.272} C_VEL
LIN {X 0,Y 569.383,Z 661.745,A -85,B 0,C 180,E1 27497.974,E2 27497.974} C_VEL
LIN {X 0,Y 569.373,Z 661.745,A -85,B 0,C 180,E1 27497.652,E2 27497.652} C_VEL
LIN {X 0,Y 568.363,Z 661.872,A -85,B 0,C 180,E1 27496.877,E2 27496.877} C_VEL
LIN {X 0,Y 561.951,Z 662.67,A -85,B 0,C 180,E1 27494.7,E2 27494.7} C_VEL
LIN {X 0,Y 561.427,Z 662.735,A -85,B 0,C 180,E1 27494.134,E2 27494.134} C_VEL
LIN {X 0,Y 561.433,Z 662.734,A -85,B 0,C 180,E1 27490.807,E2 27490.807} C_VEL
LIN {X 0,Y 561.44,Z 662.728,A -85,B 0,C 180,E1 27487.395,E2 27487.395} C_VEL
LIN {X 0,Y 561.432,Z 662.73,A -85,B 0,C 180,E1 27484.091,E2 27484.091} C_VEL
LIN {X 0,Y 561.447,Z 662.727,A -85,B 0,C 180,E1 27480.858,E2 27480.858} C_VEL
LIN {X 0,Y 561.428,Z 662.733,A -85,B 0,C 180,E1 27477.51,E2 27477.51} C_VEL
LIN {X 0,Y 561.433,Z 662.732,A -85,B 0,C 180,E1 27474.182,E2 27474.182} C_VEL
LIN {X 0,Y 561.444,Z 662.73,A -85,B 0,C 180,E1 27470.758,E2 27470.758} C_VEL
LIN {X 0,Y 561.432,Z 662.73,A -85,B 0,C 180,E1 27467.411,E2 27467.411} C_VEL
LIN {X 0,Y 561.426,Z 662.728,A -85,B 0,C 180,E1 27464.124,E2 27464.124} C_VEL
LIN {X 0,Y 561.44,Z 662.734,A -85,B 0,C 180,E1 27460.883,E2 27460.883} C_VEL
LIN {X 0,Y 561.443,Z 662.73,A -85,B 0,C 180,E1 27457.471,E2 27457.471} C_VEL
LIN {X 0,Y 561.436,Z 662.728,A -85,B 0,C 180,E1 27454.086,E2 27454.086} C_VEL
LIN {X 0,Y 561.432,Z 662.734,A -85,B 0,C 180,E1 27450.716,E2 27450.716} C_VEL
LIN {X 0,Y 561.428,Z 662.733,A -85,B 0,C 180,E1 27447.45,E2 27447.45} C_VEL
LIN {X 0,Y 561.427,Z 662.732,A -85,B 0,C 180,E1 27444.175,E2 27444.175} C_VEL
LIN {X 0,Y 561.431,Z 662.732,A -85,B 0,C 180,E1 27440.881,E2 27440.881} C_VEL
LIN {X 0,Y 561.44,Z 662.732,A -85,B 0,C 180,E1 27437.453,E2 27437.453} C_VEL
LIN {X 0,Y 561.431,Z 662.735,A -85,B 0,C 180,E1 27434.097,E2 27434.097} C_VEL
LIN {X 0,Y 561.436,Z 662.734,A -85,B 0,C 180,E1 27430.765,E2 27430.765} C_VEL
LIN {X 0,Y 561.428,Z 662.734,A -85,B 0,C 180,E1 27427.488,E2 27427.488} C_VEL
LIN {X 0,Y 561.436,Z 662.732,A -85,B 0,C 180,E1 27424.132,E2 27424.132} C_VEL
LIN {X 0,Y 561.446,Z 662.731,A -85,B 0,C 180,E1 27420.678,E2 27420.678} C_VEL
LIN {X 0,Y 561.427,Z 662.72,A -85,B 0,C 180,E1 27417.343,E2 27417.343} C_VEL
LIN {X 0,Y 561.425,Z 662.723,A -85,B 0,C 180,E1 27414.13,E2 27414.13} C_VEL
LIN {X 0,Y 561.436,Z 662.724,A -85,B 0,C 180,E1 27410.919,E2 27410.919} C_VEL
LIN {X 0,Y 561.452,Z 662.784,A -85,B 0,C 180,E1 27408.416,E2 27408.416} C_VEL
LIN {X 0,Y 570.93,Z 688.043,A -85,B 0,C 180,E1 27405.392,E2 27405.392} C_VEL
LIN {X 0,Y 579.199,Z 711.921,A -85,B 0,C 180,E1 27402.723,E2 27402.723} C_VEL
LIN {X 0,Y 579.409,Z 714.279,A -85,B 0,C 180,E1 27402.509,E2 27402.509} C_VEL
LIN {X 0,Y 576.901,Z 751.417,A -85,B 0,C 180,E1 27399.535,E2 27399.535} C_VEL
LIN {X 0,Y 573.889,Z 796.799,A -85,B 0,C 180,E1 27395.956,E2 27395.956} C_VEL
LIN {X 0,Y 571.073,Z 844.077,A -85,B 0,C 180,E1 27392.278,E2 27392.278} C_VEL
LIN {X 0,Y 568.656,Z 891.143,A -85,B 0,C 180,E1 27388.673,E2 27388.673} C_VEL
LIN {X 0,Y 568.157,Z 903.649,A -85,B 0,C 180,E1 27387.757,E2 27387.757} C_VEL
LIN {X 0,Y 569.028,Z 912.826,A -85,B 0,C 180,E1 27387.565,E2 27387.565} C_VEL
LIN {X 0,Y 565.949,Z 1048.294,A -85,B 0,C 180,E1 27385.286,E2 27385.286} C_VEL
LIN {X 0,Y 565.597,Z 1065.493,A -85,B 0,C 180,E1 27384.797,E2 27384.797} C_VEL
LIN {X 0,Y 565.117,Z 1080.748,A -85,B 0,C 180,E1 27384.18,E2 27384.18} C_VEL
LIN {X 0,Y 564.468,Z 1096.445,A -85,B 0,C 180,E1 27383.332,E2 27383.332} C_VEL
LIN {X 0,Y 563.814,Z 1110.499,A -85,B 0,C 180,E1 27382.359,E2 27382.359} C_VEL
LIN {X 0,Y 563.118,Z 1123.944,A -85,B 0,C 180,E1 27381.188,E2 27381.188} C_VEL
LIN {X 0,Y 562.505,Z 1135.342,A -85,B 0,C 180,E1 27379.956,E2 27379.956} C_VEL
LIN {X 0,Y 561.902,Z 1146.352,A -85,B 0,C 180,E1 27378.466,E2 27378.466} C_VEL
LIN {X 0,Y 561.454,Z 1154.957,A -85,B 0,C 180,E1 27376.982,E2 27376.982} C_VEL
LIN {X 0,Y 561.132,Z 1162.056,A -85,B 0,C 180,E1 27375.397,E2 27375.397} C_VEL
LIN {X 0,Y 560.943,Z 1167.213,A -85,B 0,C 180,E1 27373.819,E2 27373.819} C_VEL
LIN {X 0,Y 560.84,Z 1171.016,A -85,B 0,C 180,E1 27372.04,E2 27372.04} C_VEL
LIN {X 0,Y 560.832,Z 1172.732,A -85,B 0,C 180,E1 27370.374,E2 27370.374} C_VEL
LIN {X 0,Y 560.915,Z 1172.684,A -85,B 0,C 180,E1 27368.612,E2 27368.612} C_VEL
LIN {X 0,Y 561.065,Z 1170.875,A -85,B 0,C 180,E1 27366.961,E2 27366.961} C_VEL
LIN {X 0,Y 561.361,Z 1167.079,A -85,B 0,C 180,E1 27365.212,E2 27365.212} C_VEL
LIN {X 0,Y 561.779,Z 1161.573,A -85,B 0,C 180,E1 27363.572,E2 27363.572} C_VEL
LIN {X 0,Y 562.372,Z 1154.085,A -85,B 0,C 180,E1 27361.936,E2 27361.936} C_VEL
LIN {X 0,Y 563.118,Z 1144.817,A -85,B 0,C 180,E1 27360.407,E2 27360.407} C_VEL
LIN {X 0,Y 563.927,Z 1134.766,A -85,B 0,C 180,E1 27359.086,E2 27359.086} C_VEL
LIN {X 0,Y 564.865,Z 1122.172,A -85,B 0,C 180,E1 27357.768,E2 27357.768} C_VEL
LIN {X 0,Y 565.715,Z 1109.549,A -85,B 0,C 180,E1 27356.707,E2 27356.707} C_VEL
LIN {X 0,Y 566.572,Z 1095.198,A -85,B 0,C 180,E1 27355.749,E2 27355.749} C_VEL
LIN {X 0,Y 567.291,Z 1080.643,A -85,B 0,C 180,E1 27354.995,E2 27354.995} C_VEL
LIN {X 0,Y 567.865,Z 1064.396,A -85,B 0,C 180,E1 27354.367,E2 27354.367} C_VEL
LIN {X 0,Y 568.224,Z 1047.215,A -85,B 0,C 180,E1 27353.917,E2 27353.917} C_VEL
LIN {X 0,Y 574.614,Z 915.599,A -85,B 0,C 180,E1 27351.116,E2 27351.116} C_VEL
LIN {X 0,Y 579.304,Z 869.072,A -85,B 0,C 180,E1 27347.203,E2 27347.203} C_VEL
LIN {X 0,Y 584.528,Z 827.626,A -85,B 0,C 180,E1 27343.605,E2 27343.605} C_VEL
LIN {X 0,Y 590.822,Z 787.682,A -85,B 0,C 180,E1 27340.01,E2 27340.01} C_VEL
LIN {X 0,Y 596.77,Z 756.903,A -85,B 0,C 180,E1 27337.125,E2 27337.125} C_VEL
LIN {X 0,Y 599.936,Z 741.523,A -85,B 0,C 180,E1 27335.586,E2 27335.586} C_VEL
LIN {X 0,Y 597.181,Z 731.682,A -85,B 0,C 180,E1 27333.603,E2 27333.603} C_VEL
LIN {X 0,Y 594.836,Z 724.241,A -85,B 0,C 180,E1 27331.704,E2 27331.704} C_VEL
LIN {X 0,Y 593.155,Z 719.04,A -85,B 0,C 180,E1 27329.956,E2 27329.956} C_VEL
LIN {X 0,Y 592.294,Z 716.042,A -85,B 0,C 180,E1 27328.557,E2 27328.557} C_VEL
LIN {X 0,Y 591.813,Z 713.34,A -85,B 0,C 180,E1 27326.346,E2 27326.346} C_VEL
LIN {X 0,Y 592.153,Z 713.211,A -85,B 0,C 180,E1 27324.808,E2 27324.808} C_VEL
LIN {X 0,Y 592.901,Z 715.964,A -85,B 0,C 180,E1 27322.861,E2 27322.861} C_VEL
LIN {X 0,Y 593.853,Z 717.694,A -85,B 0,C 180,E1 27321.957,E2 27321.957} C_VEL
LIN {X 0,Y 595.52,Z 722.14,A -85,B 0,C 180,E1 27320.48,E2 27320.48} C_VEL
LIN {X 0,Y 597.533,Z 727.63,A -85,B 0,C 180,E1 27319.134,E2 27319.134} C_VEL
LIN {X 0,Y 599.341,Z 733.714,A -85,B 0,C 180,E1 27317.971,E2 27317.971} C_VEL
LIN {X 0,Y 592.111,Z 764.939,A -85,B 0,C 180,E1 27315.584,E2 27315.584} C_VEL
LIN {X 0,Y 586.576,Z 798.454,A -85,B 0,C 180,E1 27313.119,E2 27313.119} C_VEL
LIN {X 0,Y 585.304,Z 820.152,A -85,B 0,C 180,E1 27311.448,E2 27311.448} C_VEL
LIN {X 0,Y 586.155,Z 837.821,A -85,B 0,C 180,E1 27310.01,E2 27310.01} C_VEL
LIN {X 0,Y 589.034,Z 854.406,A -85,B 0,C 180,E1 27308.583,E2 27308.583} C_VEL
LIN {X 0,Y 593.632,Z 868.993,A -85,B 0,C 180,E1 27307.263,E2 27307.263} C_VEL
LIN {X 0,Y 599.959,Z 882.514,A -85,B 0,C 180,E1 27305.988,E2 27305.988} C_VEL
LIN {X 0,Y 608.322,Z 895.331,A -85,B 0,C 180,E1 27304.73,E2 27304.73} C_VEL
LIN {X 0,Y 617.401,Z 905.954,A -85,B 0,C 180,E1 27303.65,E2 27303.65} C_VEL
LIN {X 0,Y 622.837,Z 911.52,A -85,B 0,C 180,E1 27303.079,E2 27303.079} C_VEL
LIN {X 0,Y 609.254,Z 933.187,A -85,B 0,C 180,E1 27302.455,E2 27302.455} C_VEL
LIN {X 0,Y 599.313,Z 951.898,A -85,B 0,C 180,E1 27301.815,E2 27301.815} C_VEL
LIN {X 0,Y 590.471,Z 971.418,A -85,B 0,C 180,E1 27301.062,E2 27301.062} C_VEL
LIN {X 0,Y 583.371,Z 988.349,A -85,B 0,C 180,E1 27300.371,E2 27300.371} C_VEL
LIN {X 0,Y 579.132,Z 1001.12,A -85,B 0,C 180,E1 27299.821,E2 27299.821} C_VEL
LIN {X 0,Y 576.758,Z 1023.177,A -85,B 0,C 180,E1 27299.6,E2 27299.6} C_VEL
LIN {X 0,Y 575.686,Z 1062.832,A -85,B 0,C 180,E1 27299.012,E2 27299.012} C_VEL
LIN {X 0,Y 574.7,Z 1084.937,A -85,B 0,C 180,E1 27298.508,E2 27298.508} C_VEL
LIN {X 0,Y 573.458,Z 1106.702,A -85,B 0,C 180,E1 27297.828,E2 27297.828} C_VEL
LIN {X 0,Y 572.025,Z 1128.236,A -85,B 0,C 180,E1 27296.967,E2 27296.967} C_VEL
LIN {X 0,Y 570.521,Z 1148.641,A -85,B 0,C 180,E1 27295.962,E2 27295.962} C_VEL
LIN {X 0,Y 568.944,Z 1168.438,A -85,B 0,C 180,E1 27294.779,E2 27294.779} C_VEL
LIN {X 0,Y 567.353,Z 1186.861,A -85,B 0,C 180,E1 27293.47,E2 27293.47} C_VEL
LIN {X 0,Y 565.755,Z 1205.664,A -85,B 0,C 180,E1 27291.895,E2 27291.895} C_VEL
LIN {X 0,Y 564.381,Z 1221.782,A -85,B 0,C 180,E1 27290.317,E2 27290.317} C_VEL
LIN {X 0,Y 563.176,Z 1236.46,A -85,B 0,C 180,E1 27288.636,E2 27288.636} C_VEL
LIN {X 0,Y 562.191,Z 1249.83,A -85,B 0,C 180,E1 27286.851,E2 27286.851} C_VEL
LIN {X 0,Y 561.377,Z 1261.927,A -85,B 0,C 180,E1 27284.965,E2 27284.965} C_VEL
LIN {X 0,Y 560.799,Z 1272.621,A -85,B 0,C 180,E1 27282.981,E2 27282.981} C_VEL
LIN {X 0,Y 560.387,Z 1281.865,A -85,B 0,C 180,E1 27280.901,E2 27280.901} C_VEL
LIN {X 0,Y 560.179,Z 1289.646,A -85,B 0,C 180,E1 27278.725,E2 27278.725} C_VEL
LIN {X 0,Y 560.085,Z 1295.338,A -85,B 0,C 180,E1 27276.662,E2 27276.662} C_VEL
LIN {X 0,Y 560.076,Z 1299.363,A -85,B 0,C 180,E1 27274.606,E2 27274.606} C_VEL
LIN {X 0,Y 560.089,Z 1302.039,A -85,B 0,C 180,E1 27272.454,E2 27272.454} C_VEL
LIN {X 0,Y 560.102,Z 1302.992,A -85,B 0,C 180,E1 27270.408,E2 27270.408} C_VEL
LIN {X 0,Y 560.109,Z 1302.355,A -85,B 0,C 180,E1 27268.157,E2 27268.157} C_VEL
LIN {X 0,Y 560.084,Z 1300.279,A -85,B 0,C 180,E1 27266.109,E2 27266.109} C_VEL
LIN {X 0,Y 560.092,Z 1296.55,A -85,B 0,C 180,E1 27264.055,E2 27264.055} C_VEL
LIN {X 0,Y 560.153,Z 1291.015,A -85,B 0,C 180,E1 27261.892,E2 27261.892} C_VEL
LIN {X 0,Y 560.304,Z 1284.006,A -85,B 0,C 180,E1 27259.823,E2 27259.823} C_VEL
LIN {X 0,Y 560.603,Z 1275.344,A -85,B 0,C 180,E1 27257.8,E2 27257.8} C_VEL
LIN {X 0,Y 561.086,Z 1264.783,A -85,B 0,C 180,E1 27255.762,E2 27255.762} C_VEL
LIN {X 0,Y 561.758,Z 1253.147,A -85,B 0,C 180,E1 27253.878,E2 27253.878} C_VEL
LIN {X 0,Y 562.61,Z 1240.096,A -85,B 0,C 180,E1 27252.093,E2 27252.093} C_VEL
LIN {X 0,Y 563.733,Z 1224.375,A -85,B 0,C 180,E1 27250.251,E2 27250.251} C_VEL
LIN {X 0,Y 565.176,Z 1205.776,A -85,B 0,C 180,E1 27248.407,E2 27248.407} C_VEL
LIN {X 0,Y 566.665,Z 1187.015,A -85,B 0,C 180,E1 27246.827,E2 27246.827} C_VEL
LIN {X 0,Y 568.22,Z 1167.971,A -85,B 0,C 180,E1 27245.462,E2 27245.462} C_VEL
LIN {X 0,Y 569.745,Z 1147.96,A -85,B 0,C 180,E1 27244.255,E2 27244.255} C_VEL
LIN {X 0,Y 571.269,Z 1126.996,A -85,B 0,C 180,E1 27243.209,E2 27243.209} C_VEL
LIN {X 0,Y 572.713,Z 1105.344,A -85,B 0,C 180,E1 27242.327,E2 27242.327} C_VEL
LIN {X 0,Y 574.024,Z 1082.612,A -85,B 0,C 180,E1 27241.608,E2 27241.608} C_VEL
LIN {X 0,Y 575.123,Z 1058.909,A -85,B 0,C 180,E1 27241.064,E2 27241.064} C_VEL
LIN {X 0,Y 575.875,Z 1028.007,A -85,B 0,C 180,E1 27240.595,E2 27240.595} C_VEL
LIN {X 0,Y 576.834,Z 1014.678,A -85,B 0,C 180,E1 27240.422,E2 27240.422} C_VEL
LIN {X 0,Y 583.749,Z 993.36,A -85,B 0,C 180,E1 27239.42,E2 27239.42} C_VEL
LIN {X 0,Y 590.752,Z 976.264,A -85,B 0,C 180,E1 27238.692,E2 27238.692} C_VEL
LIN {X 0,Y 597.024,Z 962.75,A -85,B 0,C 180,E1 27238.158,E2 27238.158} C_VEL
LIN {X 0,Y 605.743,Z 944.947,A -85,B 0,C 180,E1 27237.494,E2 27237.494} C_VEL
LIN {X 0,Y 617.296,Z 925.291,A -85,B 0,C 180,E1 27236.87,E2 27236.87} C_VEL
LIN {X 0,Y 624.745,Z 913.656,A -85,B 0,C 180,E1 27236.543,E2 27236.543} C_VEL
LIN {X 0,Y 613.852,Z 902.211,A -85,B 0,C 180,E1 27235.345,E2 27235.345} C_VEL
LIN {X 0,Y 604.445,Z 889.042,A -85,B 0,C 180,E1 27234.071,E2 27234.071} C_VEL
LIN {X 0,Y 597.065,Z 874.964,A -85,B 0,C 180,E1 27232.802,E2 27232.802} C_VEL
LIN {X 0,Y 591.245,Z 859.034,A -85,B 0,C 180,E1 27231.459,E2 27231.459} C_VEL
LIN {X 0,Y 587.272,Z 841.313,A -85,B 0,C 180,E1 27230.067,E2 27230.067} C_VEL
LIN {X 0,Y 585.34,Z 823.065,A -85,B 0,C 180,E1 27228.731,E2 27228.731} C_VEL
LIN {X 0,Y 585.141,Z 800.876,A -85,B 0,C 180,E1 27227.214,E2 27227.214} C_VEL
LIN {X 0,Y 590.309,Z 736.924,A -85,B 0,C 180,E1 27223.109,E2 27223.109} C_VEL
LIN {X 0,Y 590.973,Z 728.113,A -85,B 0,C 180,E1 27222.527,E2 27222.527} C_VEL
LIN {X 0,Y 579.619,Z 702.272,A -85,B 0,C 180,E1 27219.664,E2 27219.664} C_VEL
LIN {X 0,Y 575.307,Z 692.764,A -85,B 0,C 180,E1 27218.523,E2 27218.523} C_VEL
LIN {X 0,Y 577.283,Z 692.883,A -85,B 0,C 180,E1 27218.153,E2 27218.153} C_VEL
LIN {X 0,Y 580.472,Z 702.309,A -85,B 0,C 180,E1 27216.584,E2 27216.584} C_VEL
LIN {X 0,Y 583.293,Z 713.508,A -85,B 0,C 180,E1 27215.048,E2 27215.048} C_VEL
LIN {X 0,Y 585.213,Z 718.173,A -85,B 0,C 180,E1 27214.695,E2 27214.695} C_VEL
LIN {X 0,Y 588.443,Z 736.216,A -85,B 0,C 180,E1 27213.857,E2 27213.857} C_VEL
LIN {X 0,Y 588.63,Z 739.655,A -85,B 0,C 180,E1 27213.748,E2 27213.748} C_VEL
LIN {X 0,Y 582.835,Z 837.945,A -85,B 0,C 180,E1 27211.926,E2 27211.926} C_VEL
LIN {X 0,Y 578.976,Z 929.957,A -85,B 0,C 180,E1 27210.348,E2 27210.348} C_VEL
LIN {X 0,Y 576.34,Z 1015.603,A -85,B 0,C 180,E1 27208.967,E2 27208.967} C_VEL
LIN {X 0,Y 575.39,Z 1038.336,A -85,B 0,C 180,E1 27208.406,E2 27208.406} C_VEL
LIN {X 0,Y 574.245,Z 1059.705,A -85,B 0,C 180,E1 27207.704,E2 27207.704} C_VEL
LIN {X 0,Y 572.821,Z 1082.135,A -85,B 0,C 180,E1 27206.767,E2 27206.767} C_VEL
LIN {X 0,Y 571.443,Z 1101.304,A -85,B 0,C 180,E1 27205.786,E2 27205.786} C_VEL
LIN {X 0,Y 569.855,Z 1121.023,A -85,B 0,C 180,E1 27204.573,E2 27204.573} C_VEL
LIN {X 0,Y 568.25,Z 1139.529,A -85,B 0,C 180,E1 27203.213,E2 27203.213} C_VEL
LIN {X 0,Y 566.656,Z 1157.073,A -85,B 0,C 180,E1 27201.696,E2 27201.696} C_VEL
LIN {X 0,Y 565.289,Z 1172.167,A -85,B 0,C 180,E1 27200.177,E2 27200.177} C_VEL
LIN {X 0,Y 563.927,Z 1187.22,A -85,B 0,C 180,E1 27198.398,E2 27198.398} C_VEL
LIN {X 0,Y 562.805,Z 1199.971,A -85,B 0,C 180,E1 27196.621,E2 27196.621} C_VEL
LIN {X 0,Y 561.837,Z 1212.066,A -85,B 0,C 180,E1 27194.638,E2 27194.638} C_VEL
LIN {X 0,Y 561.126,Z 1222.181,A -85,B 0,C 180,E1 27192.661,E2 27192.661} C_VEL
LIN {X 0,Y 560.619,Z 1230.809,A -85,B 0,C 180,E1 27190.586,E2 27190.586} C_VEL
LIN {X 0,Y 560.275,Z 1237.995,A -85,B 0,C 180,E1 27188.415,E2 27188.415} C_VEL
LIN {X 0,Y 560.098,Z 1243.443,A -85,B 0,C 180,E1 27186.252,E2 27186.252} C_VEL
LIN {X 0,Y 560.003,Z 1247.192,A -85,B 0,C 180,E1 27184.096,E2 27184.096} C_VEL
LIN {X 0,Y 559.968,Z 1249.316,A -85,B 0,C 180,E1 27181.944,E2 27181.944} C_VEL
LIN {X 0,Y 559.974,Z 1249.961,A -85,B 0,C 180,E1 27179.795,E2 27179.795} C_VEL
LIN {X 0,Y 559.967,Z 1248.995,A -85,B 0,C 180,E1 27177.646,E2 27177.646} C_VEL
LIN {X 0,Y 560.005,Z 1246.322,A -85,B 0,C 180,E1 27175.391,E2 27175.391} C_VEL
LIN {X 0,Y 560.105,Z 1242.191,A -85,B 0,C 180,E1 27173.234,E2 27173.234} C_VEL
LIN {X 0,Y 560.277,Z 1236.64,A -85,B 0,C 180,E1 27171.171,E2 27171.171} C_VEL
LIN {X 0,Y 560.609,Z 1229.458,A -85,B 0,C 180,E1 27169.102,E2 27169.102} C_VEL
LIN {X 0,Y 561.143,Z 1220.571,A -85,B 0,C 180,E1 27167.025,E2 27167.025} C_VEL
LIN {X 0,Y 561.873,Z 1210.237,A -85,B 0,C 180,E1 27165.046,E2 27165.046} C_VEL
LIN {X 0,Y 562.804,Z 1198.579,A -85,B 0,C 180,E1 27163.167,E2 27163.167} C_VEL
LIN {X 0,Y 563.938,Z 1185.703,A -85,B 0,C 180,E1 27161.388,E2 27161.388} C_VEL
LIN {X 0,Y 565.337,Z 1170.557,A -85,B 0,C 180,E1 27159.609,E2 27159.609} C_VEL
LIN {X 0,Y 566.78,Z 1154.865,A -85,B 0,C 180,E1 27158.037,E2 27158.037} C_VEL
LIN {X 0,Y 568.492,Z 1136.541,A -85,B 0,C 180,E1 27156.468,E2 27156.468} C_VEL
LIN {X 0,Y 570.087,Z 1118.846,A -85,B 0,C 180,E1 27155.176,E2 27155.176} C_VEL
LIN {X 0,Y 571.738,Z 1099.045,A -85,B 0,C 180,E1 27153.962,E2 27153.962} C_VEL
LIN {X 0,Y 573.203,Z 1079.619,A -85,B 0,C 180,E1 27152.973,E2 27152.973} C_VEL
LIN {X 0,Y 574.665,Z 1057.804,A -85,B 0,C 180,E1 27152.064,E2 27152.064} C_VEL
LIN {X 0,Y 575.864,Z 1036.18,A -85,B 0,C 180,E1 27151.354,E2 27151.354} C_VEL
LIN {X 0,Y 576.839,Z 1013.639,A -85,B 0,C 180,E1 27150.812,E2 27150.812} C_VEL
LIN {X 0,Y 577.605,Z 985.641,A -85,B 0,C 180,E1 27150.363,E2 27150.363} C_VEL
LIN {X 0,Y 582.64,Z 779.244,A -85,B 0,C 180,E1 27147.4,E2 27147.4} C_VEL
LIN {X 0,Y 583.692,Z 736.138,A -85,B 0,C 180,E1 27146.755,E2 27146.755} C_VEL
LIN {X 0,Y 577.411,Z 708.57,A -85,B 0,C 180,E1 27145.913,E2 27145.913} C_VEL
LIN {X 0,Y 575.141,Z 703.816,A -85,B 0,C 180,E1 27145.67,E2 27145.67} C_VEL
LIN {X 0,Y 568.255,Z 682.461,A -85,B 0,C 180,E1 27143.189,E2 27143.189} C_VEL
LIN {X 0,Y 561.437,Z 662.732,A -85,B 0,C 180,E1 27140.817,E2 27140.817} C_VEL
LIN {X 0,Y 561.43,Z 662.736,A -85,B 0,C 180,E1 27137.505,E2 27137.505} C_VEL
LIN {X 0,Y 561.427,Z 662.735,A -85,B 0,C 180,E1 27134.278,E2 27134.278} C_VEL
LIN {X 0,Y 561.427,Z 662.735,A -85,B 0,C 180,E1 27134.134,E2 27134.134} C_VEL
LIN {X 0,Y 560.452,Z 662.861,A -85,B 0,C 180,E1 27133.348,E2 27133.348} C_VEL
LIN {X 0,Y 553.951,Z 663.669,A -85,B 0,C 180,E1 27131.083,E2 27131.083} C_VEL
LIN {X 0,Y 553.506,Z 663.721,A -85,B 0,C 180,E1 27130.565,E2 27130.565} C_VEL
LIN {X 0,Y 553.492,Z 663.717,A -85,B 0,C 180,E1 27127.186,E2 27127.186} C_VEL
LIN {X 0,Y 553.49,Z 663.719,A -85,B 0,C 180,E1 27123.933,E2 27123.933} C_VEL
LIN {X 0,Y 553.496,Z 663.717,A -85,B 0,C 180,E1 27120.627,E2 27120.627} C_VEL
LIN {X 0,Y 553.499,Z 663.724,A -85,B 0,C 180,E1 27117.277,E2 27117.277} C_VEL
LIN {X 0,Y 553.504,Z 663.722,A -85,B 0,C 180,E1 27113.87,E2 27113.87} C_VEL
LIN {X 0,Y 553.503,Z 663.722,A -85,B 0,C 180,E1 27110.406,E2 27110.406} C_VEL
LIN {X 0,Y 553.489,Z 663.721,A -85,B 0,C 180,E1 27107.127,E2 27107.127} C_VEL
LIN {X 0,Y 553.492,Z 663.715,A -85,B 0,C 180,E1 27103.797,E2 27103.797} C_VEL
LIN {X 0,Y 553.501,Z 663.719,A -85,B 0,C 180,E1 27100.409,E2 27100.409} C_VEL
LIN {X 0,Y 553.491,Z 663.72,A -85,B 0,C 180,E1 27096.953,E2 27096.953} C_VEL
LIN {X 0,Y 553.489,Z 663.719,A -85,B 0,C 180,E1 27093.626,E2 27093.626} C_VEL
LIN {X 0,Y 553.511,Z 663.713,A -85,B 0,C 180,E1 27090.208,E2 27090.208} C_VEL
LIN {X 0,Y 553.496,Z 663.719,A -85,B 0,C 180,E1 27086.791,E2 27086.791} C_VEL
LIN {X 0,Y 553.507,Z 663.723,A -85,B 0,C 180,E1 27083.467,E2 27083.467} C_VEL
LIN {X 0,Y 553.491,Z 663.724,A -85,B 0,C 180,E1 27080.12,E2 27080.12} C_VEL
LIN {X 0,Y 553.494,Z 663.722,A -85,B 0,C 180,E1 27076.738,E2 27076.738} C_VEL
LIN {X 0,Y 553.504,Z 663.72,A -85,B 0,C 180,E1 27073.31,E2 27073.31} C_VEL
LIN {X 0,Y 553.492,Z 663.717,A -85,B 0,C 180,E1 27069.928,E2 27069.928} C_VEL
LIN {X 0,Y 553.49,Z 663.722,A -85,B 0,C 180,E1 27066.584,E2 27066.584} C_VEL
LIN {X 0,Y 553.502,Z 663.719,A -85,B 0,C 180,E1 27063.27,E2 27063.27} C_VEL
LIN {X 0,Y 553.507,Z 663.725,A -85,B 0,C 180,E1 27059.857,E2 27059.857} C_VEL
LIN {X 0,Y 553.493,Z 663.722,A -85,B 0,C 180,E1 27056.388,E2 27056.388} C_VEL
LIN {X 0,Y 553.505,Z 663.721,A -85,B 0,C 180,E1 27052.984,E2 27052.984} C_VEL
LIN {X 0,Y 553.506,Z 663.728,A -85,B 0,C 180,E1 27049.572,E2 27049.572} C_VEL
LIN {X 0,Y 553.49,Z 663.734,A -85,B 0,C 180,E1 27048.985,E2 27048.985} C_VEL
LIN {X 0,Y 563.085,Z 689.12,A -85,B 0,C 180,E1 27045.889,E2 27045.889} C_VEL
LIN {X 0,Y 571.121,Z 712.153,A -85,B 0,C 180,E1 27043.258,E2 27043.258} C_VEL
LIN {X 0,Y 572.294,Z 716.545,A -85,B 0,C 180,E1 27042.796,E2 27042.796} C_VEL
LIN {X 0,Y 569.695,Z 753.108,A -85,B 0,C 180,E1 27039.839,E2 27039.839} C_VEL
LIN {X 0,Y 566.577,Z 798.349,A -85,B 0,C 180,E1 27036.243,E2 27036.243} C_VEL
LIN {X 0,Y 563.688,Z 844.882,A -85,B 0,C 180,E1 27032.591,E2 27032.591} C_VEL
LIN {X 0,Y 561.129,Z 892.124,A -85,B 0,C 180,E1 27028.934,E2 27028.934} C_VEL
LIN {X 0,Y 560.599,Z 904.251,A -85,B 0,C 180,E1 27028.032,E2 27028.032} C_VEL
LIN {X 0,Y 561.491,Z 913.711,A -85,B 0,C 180,E1 27027.83,E2 27027.83} C_VEL
LIN {X 0,Y 558.247,Z 1049.04,A -85,B 0,C 180,E1 27025.496,E2 27025.496} C_VEL
LIN {X 0,Y 557.893,Z 1065.54,A -85,B 0,C 180,E1 27025.023,E2 27025.023} C_VEL
LIN {X 0,Y 557.374,Z 1081.568,A -85,B 0,C 180,E1 27024.369,E2 27024.369} C_VEL
LIN {X 0,Y 556.69,Z 1097.373,A -85,B 0,C 180,E1 27023.5,E2 27023.5} C_VEL
LIN {X 0,Y 556.014,Z 1111.283,A -85,B 0,C 180,E1 27022.522,E2 27022.522} C_VEL
LIN {X 0,Y 555.284,Z 1124.787,A -85,B 0,C 180,E1 27021.33,E2 27021.33} C_VEL
LIN {X 0,Y 554.644,Z 1136.168,A -85,B 0,C 180,E1 27020.083,E2 27020.083} C_VEL
LIN {X 0,Y 554.031,Z 1146.808,A -85,B 0,C 180,E1 27018.629,E2 27018.629} C_VEL
LIN {X 0,Y 553.56,Z 1155.533,A -85,B 0,C 180,E1 27017.123,E2 27017.123} C_VEL
LIN {X 0,Y 553.211,Z 1162.706,A -85,B 0,C 180,E1 27015.516,E2 27015.516} C_VEL
LIN {X 0,Y 553.008,Z 1167.974,A -85,B 0,C 180,E1 27013.915,E2 27013.915} C_VEL
LIN {X 0,Y 552.897,Z 1171.849,A -85,B 0,C 180,E1 27012.11,E2 27012.11} C_VEL
LIN {X 0,Y 552.89,Z 1173.677,A -85,B 0,C 180,E1 27010.419,E2 27010.419} C_VEL
LIN {X 0,Y 552.978,Z 1173.709,A -85,B 0,C 180,E1 27008.632,E2 27008.632} C_VEL
LIN {X 0,Y 553.143,Z 1172.009,A -85,B 0,C 180,E1 27006.956,E2 27006.956} C_VEL
LIN {X 0,Y 553.456,Z 1168.297,A -85,B 0,C 180,E1 27005.183,E2 27005.183} C_VEL
LIN {X 0,Y 553.876,Z 1163.321,A -85,B 0,C 180,E1 27003.623,E2 27003.623} C_VEL
LIN {X 0,Y 554.485,Z 1156.038,A -85,B 0,C 180,E1 27001.963,E2 27001.963} C_VEL
LIN {X 0,Y 555.208,Z 1147.792,A -85,B 0,C 180,E1 27000.516,E2 27000.516} C_VEL
LIN {X 0,Y 556.108,Z 1137.387,A -85,B 0,C 180,E1 26999.073,E2 26999.073} C_VEL
LIN {X 0,Y 557.012,Z 1126.333,A -85,B 0,C 180,E1 26997.84,E2 26997.84} C_VEL
LIN {X 0,Y 557.987,Z 1113.165,A -85,B 0,C 180,E1 26996.661,E2 26996.661} C_VEL
LIN {X 0,Y 558.826,Z 1100.381,A -85,B 0,C 180,E1 26995.742,E2 26995.742} C_VEL
LIN {X 0,Y 559.687,Z 1084.953,A -85,B 0,C 180,E1 26994.875,E2 26994.875} C_VEL
LIN {X 0,Y 560.334,Z 1069.385,A -85,B 0,C 180,E1 26994.213,E2 26994.213} C_VEL
LIN {X 0,Y 560.789,Z 1052.464,A -85,B 0,C 180,E1 26993.708,E2 26993.708} C_VEL
LIN {X 0,Y 564.828,Z 968.189,A -85,B 0,C 180,E1 26991.826,E2 26991.826} C_VEL
LIN {X 0,Y 567.714,Z 917.033,A -85,B 0,C 180,E1 26990.726,E2 26990.726} C_VEL
LIN {X 0,Y 572.692,Z 870.79,A -85,B 0,C 180,E1 26986.778,E2 26986.778} C_VEL
LIN {X 0,Y 578.402,Z 828.679,A -85,B 0,C 180,E1 26983.065,E2 26983.065} C_VEL
LIN {X 0,Y 585.205,Z 788.565,A -85,B 0,C 180,E1 26979.392,E2 26979.392} C_VEL
LIN {X 0,Y 591.29,Z 759.202,A -85,B 0,C 180,E1 26976.585,E2 26976.585} C_VEL
LIN {X 0,Y 594.13,Z 746.017,A -85,B 0,C 180,E1 26975.225,E2 26975.225} C_VEL
LIN {X 0,Y 591.699,Z 736.813,A -85,B 0,C 180,E1 26973.288,E2 26973.288} C_VEL
LIN {X 0,Y 589.793,Z 730.245,A -85,B 0,C 180,E1 26971.55,E2 26971.55} C_VEL
LIN {X 0,Y 588.363,Z 725.399,A -85,B 0,C 180,E1 26969.88,E2 26969.88} C_VEL
LIN {X 0,Y 587.585,Z 722.474,A -85,B 0,C 180,E1 26968.486,E2 26968.486} C_VEL
LIN {X 0,Y 587.266,Z 719.893,A -85,B 0,C 180,E1 26966.285,E2 26966.285} C_VEL
